// TIA Portal project "Niagara_V1" (V16)

(* hardware
DEVICE "S7-1200 station_1"  S7-1200 Station
   slot 0: "Rack_0"  S7-1200 Rack  Rack  V1.0
   slot 1: "PLC_Start"  CPU 1214C DC/DC/Rly  6ES7 214-1HG40-0XB0  V4.4
   slot 2: "DI 16x24VDC_2"  6ES7 221-1BH32-0XB0  V2.0
   slot 3: "DQ 16xRelay_1"  SM 1222 DQ16 x relay  6ES7 222-1HH32-0XB0  V2.0
   slot 3: "CB 1241 (RS485)"  CB 1241 (RS485)  6ES7 241-1CH30-1XB0  V1.0
   slot 4: "DQ 16xRelay_3"  SM 1222 DQ16 x relay  6ES7 222-1HH32-0XB0  V2.0
   slot 5: "AI 8xRTD_1"  SM 1231 AI8 x RTD  6ES7 231-5PF32-0XB0  V2.0
   slot 6: "AI 4xRTD_1"  SM 1231 AI4 x RTD  6ES7 231-5PD32-0XB0  V2.0
   slot 7: "AQ 4x14BIT_2"  6ES7 232-4HD32-0XB0  V2.1
*)

// ===== PLC "PLC_Start"  CPU 1214C DC/DC/Rly =====

VAR_GLOBAL   // PLC tag table "Default tag table"
   "rAlarm_SetMinPressSteam" AT %MW12 : Int;   // Уставка минимального давления пара
   "rAI_Press1" AT %MW14 : Int;   // Давление датчика
   "bAlarmPress1" AT %M16.0 : Bool;
   "rAlarm_SetMinPressWater" AT %MW18 : Int;   // Уставка аварийного давления воды
   "rAI_Press2" AT %MW20 : Int;
   "test_PID_P_Backup" AT %MD28 : Real;
   "testLoadBackUp" AT %M1.1 : Bool;
   "Test_eee" AT %M1.2 : Bool;
   "System_Byte" AT %MB510 : Byte;
   "FirstScan" AT %M510.0 : Bool;
   "DiagStatusUpdate" AT %M510.1 : Bool;
   "AlwaysTRUE" AT %M510.2 : Bool;
   "AlwaysFALSE" AT %M510.3 : Bool;
END_VAR

VAR_GLOBAL   // PLC tag table "HMI_"
   "bHMI_button_Start" AT %M2.0 : Bool;   // Кнопка старт
   "bHMI_button_Stop" AT %M2.1 : Bool;   // Кнопка стоп
   "bHMI_button_Pause" AT %M2.2 : Bool;   // Кнопка пауза
   "bHMI_Button_ConveyorStart" AT %M2.4 : Bool;   // Кнопка подтверждения старта конвейера
   "bStartAllowed" AT %M100.0 : Bool;   // Готовность к старту
   "bOpenWindStartConveyor" AT %M100.1 : Bool;   // Вызов окна подтверждения оператором старта конвейера
   "iHMI_Num_StatrPaster" AT %MW4 : Int;   // Статус работы пастризаора
   "sHMI_Text_State" AT %MB3 : Char;   // Ткстом статус пастеризатора
   "bTypePID_Zone1" AT %M8.0 : Bool;   // Тип ПИД - 1 - Охлаждение, 0 - Нагрев
   "bTypePID_Zone2" AT %M8.1 : Bool;   // Тип ПИД - 1 - Охлаждение, 0 - Нагрев
   "bTypePID_Zone3" AT %M8.2 : Bool;   // Тип ПИД - 1 - Охлаждение, 0 - Нагрев
   "bTypePID_Zone4" AT %M8.3 : Bool;   // Тип ПИД - 1 - Охлаждение, 0 - Нагрев
   "bTypePID_Zone5" AT %M8.4 : Bool;   // Тип ПИД - 1 - Охлаждение, 0 - Нагрев
   "rHMI_SpeedConveyor" AT %MD60 : Real;   // Расчетная Скорость конвейера
   "rHMI_TimeHoldMin" AT %MD56 : Real;   // Для удобства восприятия времени выдержки
   "bResetCommon" AT %M0.3 : Bool;   // Глобальный сброс аварий
   "bAllAuto" AT %M0.6 : Bool;   // Перевод всего оборудования в авто с ручного
   "bZoomerOff" AT %M0.7 : Bool;   // Выкл пищалка
   "bHMI_button_Start_Sterilization" AT %M2.5 : Bool;   // Кнопка старт Стерилизации
   "bHMI_Steril_Fimish" AT %M8.7 : Bool;   // Стерилизация готова флаг
   "iHMI_Steril_sec" AT %MW22 : Int;   // СЕК таймера стерилизациии
   "iHMI_Steril_min" AT %MW26 : Int;   // МИН таймера стерилизации
   "iHMIWind_FinishStiril" AT %MW32 : Int;   // Всплывающее окно на панели
   "bOpenWindSterilFinish" AT %M34.0 : Bool;   // Вызвать окно окончание стирилизации
   "bHMI_Start_Banya" AT %M8.6 : Bool;   // Кнопка старт режима "Баня"
   "bTypePID_Zone6" AT %M9.1 : Bool;   // Тип ПИД - 1 - Охлаждение, 0 - Нагрев
   "bTypePID_Zone7" AT %M9.2 : Bool;   // Тип ПИД - 1 - Охлаждение, 0 - Нагрев
   "bTypePID_Zone8" AT %M9.3 : Bool;   // Тип ПИД - 1 - Охлаждение, 0 - Нагрев
   "bTypePID_Zone9" AT %M9.4 : Bool;   // Тип ПИД - 1 - Охлаждение, 0 - Нагрев
   "bTypePID_Zone10" AT %M9.5 : Bool;   // Тип ПИД - 1 - Охлаждение, 0 - Нагрев
   "bTypePID_Zone11" AT %M9.6 : Bool;   // Тип ПИД - 1 - Охлаждение, 0 - Нагрев
   "bSafetyMode" AT %M10.3 : Bool;   // Режим защиты от перепастеризации
   "bResSafetyMode" AT %M10.4 : Bool;   // Сброс режима защиты от перепастеризации
   "bCheck_ModeSafety" AT %M10.5 : Bool;   // Галочка - разрешение работы режима защиты от перепастеризации
   "bStateZonesBanya_OK" AT %M10.6 : Bool;   // Статус готовности по зонам в режиме Баня
   "bHasPrior_Stop_Bany" AT %M10.7 : Bool;   // Установлен приоритет по стопу конвейера при отклонении в режиме Баня
   "iNomberZoneAlarmBany" AT %MW40 : Int;   // Номер зоны с отклонениями от уставок
   "rHMI_Fact_SpeedConveyor" AT %MD64 : Real;   // Фактическая Скорость конвейера
END_VAR

VAR_GLOBAL   // PLC tag table "DI"
   "E-Stop №1" AT %I0.0 : Bool;
   "E-Stop №2" AT %I0.1 : Bool;
   "E-Stop №3" AT %I0.2 : Bool;
   "Контроль фаз" AT %I2.7 : Bool;
   "Уровнь_Низ 1" AT %I2.3 : Bool;
   "Уровнь_Верх 1" AT %I2.4 : Bool;
   "Д_Затор" AT %I2.6 : Bool;
   "Частотник (работа) 1" AT %I2.0 : Bool;
   "Частотник (работа) 2" AT %I2.1 : Bool;
   "Частотник (работа) 3" AT %I2.2 : Bool;
   "Пускатель включен 1" AT %I0.3 : Bool;
   "Пускатель включен 2" AT %I0.4 : Bool;
   "Пускатель включен 3" AT %I0.5 : Bool;
   "Пускатель включен 4" AT %I0.6 : Bool;
   "Пускатель включен 5" AT %I0.7 : Bool;
   "Пускатель включен 6" AT %I1.0 : Bool;
   "Пускатель включен 7" AT %I1.1 : Bool;
   "Пускатель включен 8" AT %I1.2 : Bool;
   "Пускатель включен 9" AT %I1.3 : Bool;
   "Пускатель включен 10" AT %I1.4 : Bool;
   "Пускатель вкл Воздуходувка" AT %I1.5 : Bool;
   "Д_Коленвала" AT %I2.5 : Bool;
   "Д_Давл Воздуха" AT %I3.0 : Bool;
END_VAR

VAR_GLOBAL   // PLC tag table "MyTags"
   "rHoldtimeMIN_Out" AT %MD52 : Real;   // Время выдержки в мин
   "Разрешение работы конвейера" AT %M0.0 : Bool;   // Команда разрешения от Глобального блока работы
   "Авария, ошибка в системе" AT %M0.1 : Bool;   // Метка ошибок или аварий
   "iNomberZoneAlarm" AT %MW6 : Int;   // Номер зоны с отклонениями
   "bMain_AlarmSystem" AT %M2.3 : Bool;   // АВария в системе (Общая)
   "bStartWork_Main_TunelPaster" AT %M1.7 : Bool;   // Старт-Работа тунельного пастеризатора (ОБЩИЙ)
   "bHasPrior_Stop" AT %M10.1 : Bool;   // Имеется маркер разрешения "СТОП - конвейер
   "bStateZones_OK" AT %M10.0 : Bool;   // Все зоны готовы к работе
   "bStartFillBac_1" AT %M0.4 : Bool;   // Ком_Наполнение бака 1
   "bStartFillBac_2" AT %M0.5 : Bool;   // Ком_Наполнение бака 2
   "AlarmPress" AT %M0.2 : Bool;   // Общая авария давления
   "bStartWork_Sterilization" AT %M2.6 : Bool;   // Старт-Работа режима стерилизации
   "bState_Stiril_Zone_OK" AT %M1.0 : Bool;   // Все зоны готовы к стерилизации
   "iNumZoneStiril_NotOk" AT %MW24 : Int;   // Номер зоны не готовые стирилизации
   "bStartWork_БАНЯ" AT %M9.0 : Bool;
   "ПЕ_Вер-1" AT %M11.3 : Bool;   // Работа расчета Пе (вер_1)
END_VAR

VAR_GLOBAL   // PLC tag table "Timers_CPU"
   "Time_0.1s" AT %M500.0 : Bool;
   "Time_0.2s" AT %M500.1 : Bool;
   "Time_0.4s" AT %M500.2 : Bool;
   "Time_0.5s" AT %M500.3 : Bool;
   "Time_0.8s" AT %M500.4 : Bool;
   "Time_1s" AT %M500.5 : Bool;
   "Time_1.6s" AT %M500.6 : Bool;
   "Time_2s" AT %M500.7 : Bool;
END_VAR

VAR_GLOBAL   // PLC tag table "DO"
   "Пневмо_остров клапан 1" AT %Q0.0 : Bool;
   "Пневмо_остров клапан 2" AT %Q0.1 : Bool;
   "Пневмо_остров клапан 3" AT %Q0.2 : Bool;
   "Пневмо_остров клапан 4" AT %Q0.3 : Bool;
   "Пневмо_остров клапан 5" AT %Q0.4 : Bool;
   "Пневмо_остров клапан 6" AT %Q0.5 : Bool;
   "Пневмо_остров клапан 7" AT %Q0.6 : Bool;
   "Пневмо_остров клапан 8" AT %Q16.7 : Bool;   // Не используем выход общий с 9 клапаном
   "Пневмо_остров клапан 9" AT %Q1.0 : Bool;
   "Пневмо_остров клапан 10" AT %Q1.1 : Bool;
   "Частотник Пуск 1" AT %Q6.3 : Bool;   // Реле К 9
   "Частотник Пуск 2" AT %Q6.4 : Bool;   // Реле К 10
   "Частотник Пуск 3" AT %Q6.5 : Bool;   // Реле К 11
   "Световая колонна - зеленый" AT %Q7.0 : Bool;
   "Световая колонна - желтый" AT %Q7.1 : Bool;
   "Световая колонна - красный" AT %Q7.2 : Bool;
   "Световая колонна – звуковой сигнал" AT %Q7.3 : Bool;
   "Пускатель №1" AT %Q4.0 : Bool;
   "Пускатель №2" AT %Q4.1 : Bool;
   "Пускатель №3" AT %Q4.2 : Bool;
   "Пускатель №4" AT %Q4.3 : Bool;
   "Пускатель №5" AT %Q4.4 : Bool;
   "Пускатель №6" AT %Q4.5 : Bool;
   "Пускатель №7" AT %Q4.6 : Bool;
   "Пускатель Воздуходувка" AT %Q6.2 : Bool;
   "Пуск транспортера" AT %Q11.0 : Bool;   // Реле К 12
   "Пускатель №8" AT %Q4.7 : Bool;
   "Пускатель №9" AT %Q6.0 : Bool;
   "Пускатель №10" AT %Q6.1 : Bool;
   "Пневмо_остров клапан 11" AT %Q15.0 : Bool;   // Не используем выход общий с 12 клапаном
   "Пневмо_остров клапан 12" AT %Q5.1 : Bool;
   "КЛ_Химия-1" AT %Q5.2 : Bool;
   "КЛ_Пара" AT %Q5.5 : Bool;
   "КЛ_Стирилизации" AT %Q5.6 : Bool;
   "КЛ_Подпидки" AT %Q5.4 : Bool;
   "КЛ_Химия-2" AT %Q5.3 : Bool;
END_VAR

VAR_GLOBAL   // PLC tag table "AI"
   "TT 1" AT %IW140 : Int;   // PT100
   "TT 2" AT %IW142 : Int;   // PT100
   "TT 3" AT %IW144 : Int;   // PT100
   "TT 4" AT %IW146 : Int;   // PT100
   "TT 5" AT %IW148 : Int;   // PT100
   "TT 6" AT %IW150 : Int;   // PT100
   "TT 7" AT %IW152 : Int;   // PT100
   "TT 8" AT %IW154 : Int;   // PT100
   "AI_0.0_Датчик давления 1" AT %IW112 : Int;   // 4-20mA
   "AI_0.1_Датчик давления 2" AT %IW114 : Int;   // 4-20mA
   "AI_0.2_Датчик давления 3" AT %IW116 : Int;   // 4-20mA
   "AI_0.3_" AT %IW118 : Int;   // 4-20mA
   "TT 9" AT %IW156 : Int;
   "TT 10" AT %IW158 : Int;
END_VAR

VAR_GLOBAL   // PLC tag table "AO"
   "Упр частоты 1" AT %QW180 : Int;
   "Упр частоты 2" AT %QW182 : Int;
   "Упр частоты 3" AT %QW184 : Int;
END_VAR

VAR_GLOBAL   // PLC tag table "Alarms"
   "Ai_Alarm_1" AT %M50.0 : Bool;
   "Ai_Alarm_2" AT %M50.1 : Bool;
   "Ai_Alarm_3" AT %M50.2 : Bool;
   "Ai_Alarm_4" AT %M50.3 : Bool;
   "Ai_Alarm_5" AT %M50.4 : Bool;
   "Ai_Alarm_6" AT %M50.5 : Bool;
END_VAR

VAR_GLOBAL   // PLC tag table "__TEST"
   "bT_Alarm" AT %M1.3 : Bool;
   "bTOpenWind" AT %M1.4 : Bool;
   "iTestPause" AT %MW1 : Int;
   "bTZoomOff" AT %M8.5 : Bool;
   "Test_Time" AT %MD36 : DInt;
   "test_reset" AT %M9.7 : Bool;
   "Test_Alarm" AT %M10.2 : Bool;
   "ТестБаня" AT %M11.0 : Bool;
   "ТестБаняОк" AT %M11.1 : Bool;
   "Тест_СтартБаня" AT %M11.2 : Bool;
   "Тест_Старт ПЕ" AT %M11.4 : Bool;
   "Тест-СкоростьКонв" AT %MD42 : Real;
   "T485_MB_ADDR" AT %MW46 : UInt;
   "T485_MODE" AT %MB17 : USInt;
   "T485_DATA_ADDR" AT %MD68 : UDInt;
   "T485_DATA_LEN" AT %MW48 : UInt;
   "T485_GetData" AT %MW11 : Int;
   "T_485_REQ" AT %M16.1 : Bool;
   "MB_ADDR_T1" AT %MW72 : UInt;
   "MB_MODE_T" AT %MB35 : USInt;
   "MB_DATA_ADDR" AT %MD74 : UDInt;
   "MB_LENGH_T" AT %MW78 : UInt;
   "MB_MODE_T2" AT %MB51 : USInt;
   "MB_DATA_ADDR2" AT %MD80 : UDInt;
   "MB_LENGH_T2" AT %MW84 : UInt;
END_VAR

VAR_GLOBAL   // PLC tag table "RS-485"
   "Управляемый клапан №1" AT %MW111 : Int;
   "Управляемый клапан №2" AT %MW114 : Int;
   "Управляемый клапан №3" AT %MW116 : Int;
   "Управляемый клапан №4" AT %MW118 : Int;
   "Управляемый клапан №5" AT %MW120 : Int;
   "Управляемый клапан №6" AT %MW122 : Int;
   "Управляемый клапан №7" AT %MW124 : Int;
   "Управляемый клапан №8" AT %MW126 : Int;
   "Управляемый клапан №9" AT %MW128 : Int;
   "Управляемый клапан №10" AT %MW130 : Int;
   "Управляемый клапан №11" AT %MW132 : Int;
   "Управляемый клапан №12" AT %MW134 : Int;
END_VAR

TYPE "FV_o/c"
   STRUCT
      bOpenCmd : Bool;   // Команда открыть (автомат)
      bManualMode : Bool;   // Ручной режим (TRUE)
      bManualOpen : Bool;   // Команда открыть в ручном режиме
      bFeedbackOpen : Bool;   // Обратная связь "Открыт"
      tMaxTime : Time;   // Время на открытие
      bResetAlarm : Bool;   // Сброс аварии
      bCheckFeedback : Bool;   // Выбирается есть ли обратная связь у клапана
      bOutOpen : Bool;   // Выход на открытие клапана
      iOutState : Int;   // Выход статуса клапана
   END_STRUCT;
END_TYPE

TYPE "ZoneStatus"
   STRUCT
      bInSetpoint : Bool;   // Зона в уставке по температуре
      bOutOfRange : Bool;   // Зона вышла от уставки на > дельта
      bHasPriority : Bool;   // Зона имеет приоритет на остановку конвейера
   END_STRUCT;
END_TYPE

TYPE "Zone_Pararm"
   STRUCT
      rTemp : Real;   // Температура с датчика
      rSet : Real := 20.0;   // Уставка
      rDeltaDown : Real := 1.0;   // ДельтаНижний предел
      rDeltaUP : Real := 1.0;   // ДельтаВерхний Предел
      bPriority : Bool;   // Приоритет
      bOUT_ZoneStatus : "ZoneStatus";   // Состояние зоны_
   END_STRUCT;
END_TYPE

TYPE "FV_regul"
   STRUCT
      bHMI_ManualMode : Bool;   // Переключение режима авто/ручно (0 - А, 1 - Р)
      "bManualOpen/Close" : Bool;   // Ручн режим выход DO для клапана
      rHMI_ManualSet : Real;   // Уставка в ручном режиме (0-100)
      "bAutoOpen/Close" : Bool;   // Авто режим Сигнал DO на выход для клапана
      rAuto_Set : Real;   // Уставка в автоматическом режиме
      iOut_AO : Int;   // Сигнал на аналоговый выход
      "rHMI_Out_FV-%" : Real;   // Состояние в % (0-100)
      "bOut_DO_Open/Close" : Bool;   // Сигнал выход для DO
      bOut_State_ValveOpen : Int;   // Cтатуса - клапан открыт (1)/закрыт(0)
   END_STRUCT;
END_TYPE

TYPE "Коэф ПИД"
   STRUCT
      Set : Real;   // Уставка
      Gain : Int;   // Коэф П
      I : DInt;   // Коэф И
      D : DInt;   // Коэф Д
   END_STRUCT;
END_TYPE

TYPE "PE_Param"
   STRUCT
      rПЕ_Задан : Real;
      rДлина_Конв : Real;
      rZ_Коэф : Real := 1.393;
      rТref : Real := 60.0;
      rТемп_Мин : Real;
      rТемп_Макс : Real;
      "rСкоростьКонв_м/мин" : Real;
      rРучноеЗначТемп : Real;
      diВремяПростоя : DInt := 60000;
      bManualTemp : Bool;
   END_STRUCT;
END_TYPE

TYPE "tipe_Pumps"
   STRUCT
      bAutoMode_Work : Bool;   // автоматический режим
      bManualMode : Bool;   // Ручной режим вкл/выкл
      bManualStart : Bool;   // Старт в ручном режиме
      rManualSpeed : Real;   // Скорость в ручном режиме
      rHMI_Speed : Real;   // Выходная скороость для HMI
      bHMI_PumpRun : Bool;   // Статус работы для HMI
      bresAlarm : Bool;   // Сброс аварий
      iStatusPump : Int;   // Статус насоса
      bIn_DryRunning : Bool;   // Сигнал сухого хода
      bIn_AutomatState : Bool;   // Вход статуса состояния автоматов
      bIn_PuskatelState : Bool;   // Вход статуса состояния пускателя
      bIn_Run_Ok_State : Bool;   // Вход подтверждения старта (частотники)
   END_STRUCT;
END_TYPE

TYPE "Tipe_Conveyor"
   STRUCT
      bManualMode : Bool;   // Ручной режим вкл/выкл
      bManualStart : Bool;   // Старт в ручном режиме
      rManualSpeed : Real;   // Скорость в ручном режиме
      bresAlarm : Bool;   // Сброс аварий
      rAutoSpeed : Real;   // Автомат_Заданная скорость конвеера
      rHMI_Speed : Real;   // Выходная скороость для HMI
      bHMI_Conv_Run : Bool;   // Статус работы для HMI
      iStatusConve : Int;   // Статус конвейера
      bIn_AutomatState : Bool;   // Вход статуса состояния автоматов
      bInPuskatelState : Bool;   // Вход статуса состояния пускателя
      bInRun_Ok_State : Bool;   // Вход подтверждения старта (частотники)
   END_STRUCT;
END_TYPE

TYPE "Tipe_DI"
   STRUCT
      f_DI_out : Bool;
      "bFiltr_on/off" : Bool := true;   // Вкл/выкл фильтрацию входа
      diTime_filtr : Time := T#100ms;   // Уставка времени фильтрации
      bSimulation : Bool;   // Включение режима симуляции
      "bSim_On/Off" : Bool;   // Управление симуляцией
   END_STRUCT;
END_TYPE

TYPE "Tipe_Filling_Bac"
   STRUCT
      bManualMode : Bool;
      bManualOpen : Bool;
      diTimeCloseValve : DInt;   // Таймер задержки закрытия клапана по верхнему уровню
   END_STRUCT;
END_TYPE

TYPE "Tipe_AI"
   STRUCT
      bSimulate : Bool;   // Вкл симуляции датчика
      rSimulateValue : Real;   // Значение симуляции датчика
      rSensor_HL : Real;   // Верхний предел датчика
      rSensor_LL : Real;   // Нижний предел датчика
      bFiltr : Bool;   // Управление фильтром значений
      rAI_Value : Real;   // Значение аналогового датчика
   END_STRUCT;
END_TYPE

TYPE "tipePress"
   STRUCT
      rInPress : Real;   // Значение с датчика
      rSetpoint : Real := 2.0;   // Уставка минимального давления
      bAlarm_Press : Bool;   // Выход АВАРИЯ
   END_STRUCT;
END_TYPE

TYPE "tipePumpHim"
   STRUCT
      Чек_вРежимеПастер : Bool;   // Указание в панели на разрешения работы насоса в режиме пастеризации
      Чек_вРежимеМойка : Bool;   // Указание в панели на разрешения работы насоса в режиме Мойка
      ВремяРаботы : DInt := 5;   // Время продолжительности импульса работы насоса
      ВремяПаузы : DInt := 10;   // Время паузы между импульсами
   END_STRUCT;
END_TYPE

TYPE "StopMgr"
   STRUCT
      Timer_Stop : IEC_TIMER;   // Таймер длительности простоя
      Duration : Time;   // Длительность простоя
      PU_Stop_Add : Real;   // Доп. ПЕ, набранные на простое
      Reject_Required : Bool;   // Флаг необходимости отбраковки
   END_STRUCT;
END_TYPE

// folder: PE_V2

TYPE "Zone_Config"
   STRUCT
      Length : Real;   // Длина зоны (м)
      TempWater_Set : Real;   // Уставка температуры воды (°C)
      TempWater_Act : Real;   // Фактическая температура воды (°C)
      TimeInZone : Real;   // Расчётное время в зоне (мин)
      TempProd_In : Real;   // Т-ра продукта на входе в зону (°C)
      TempProd_Out : Real;   // Т-ра продукта на выходе из зоны (°C)
      TempProd_Avg : Real;   // Средняя Т-ра в зоне (°C)
      PU_Zone : Real;   // ПЕ, накопленные в этой зоне
      ZoneType : Bool;   // 1=Нагрев, 2=Выдержка, 3=Охлаждение
      Status_OK : Bool;   // Флаг: расчёт корректен
   END_STRUCT;
END_TYPE

TYPE "ProductPosition"
   STRUCT
      TempProduct : Real;   // Расчётная температура продукта (°C)
      PU_Accumulated : Real;   // Накопленные ПЕ для этой позиции
      InTunnel : Bool;   // Флаг: позиция занята продуктом
      ZoneIndex : Int;   // Номер текущей зоны (1-9)
   END_STRUCT;
END_TYPE

TYPE "Recipe"
   STRUCT
      ID : Int;   // ID рецепта
      "Name" : String;   // Название рецепта
      K_Coeff : Real;   // Коэффициент теплопередачи (1/мин)
      PU_Target_Min : Real;   // Минимально допустимые ПЕ
      PU_Target_Max : Real;   // Максимально допустимые ПЕ
      TempProd_Inlet : Real;   // Температура продукта на входе (°C)
      Speed_Set : Real;   // Уставка скорости ленты (м/мин)
      ZoneConfig : Array[1..9] of "Zone_Config";   // Массив зон
   END_STRUCT;
END_TYPE

TYPE "Status_V2"
   STRUCT
      PU_Total : Real;   // Итоговые ПЕ (последняя вышедшая бутылка)
      PU_Current_Avg : Real;   // Средние ПЕ продукта сейчас в туннеле
      TempProd_Max : Real;   // Макс. температура продукта в туннеле
      Speed_Act : Real;   // Фактическая скорость (м/мин)
      PosCount : Int;   // Количество активных позиций в туннеле
      Line_Run : Bool;   // Статус линии (1=работает)
   END_STRUCT;
END_TYPE

TYPE "Alarm"
   STRUCT
      Temp_Deviation : Bool;   // Отклонение температуры воды
      PU_Under : Bool;   // Недопастеризация
      PU_Over : Bool;   // Перепастеризация
      Sensor_Fault : Bool;   // Неисправность датчика
      Stop_Request : Bool;   // Запрос остановки линии
      Jam_Detected : Bool;   // Сигнал затора
   END_STRUCT;
END_TYPE

// folder: PE_V3

TYPE "ZoneDate"
   STRUCT
      TempWater_Act : Real;   // Фактическая температура воды (°C)
      TimeInZone : Real;   // Расчётное время в зоне (мин)
      TempProd_In : Real;   // Т-ра продукта на входе в зону (°C)
      TempProd_Out : Real;   // Т-ра продукта на выходе из зоны (°C)
      TempProd_Avg : Real;   // Средняя Т-ра в зоне (°C)
      PU_Zone : Real;   // ПЕ, накопленные в этой зоне
   END_STRUCT;
END_TYPE

TYPE "Status_V3"
   STRUCT
      PU_Total : Real;   // Итоговые ПЕ (последняя вышедшая бутылка)
      TempProd_Exit : Real;
      Speed_Act : Real;   // Фактическая скорость (м/мин)
      Line_Run : Bool;   // Статус линии (1=работает)
      ZoneData : Array[1..9] of "ZoneDate";   // Данные по зонам
      Calculation_Ready : Bool;   // Флаг: расчёт выполнен
   END_STRUCT;
END_TYPE

TYPE "Zone_Config_V3"
   STRUCT
      Length : Real;   // Длина зоны (м)
      TempWater_Set : Real;   // Уставка температуры воды (°C)
   END_STRUCT;
END_TYPE

// folder: (top level)

DATA_BLOCK "Test_Beep_DB"   // DB129
{ S7_Optimized_Access := 'TRUE' }
VERSION : 0.1
// stored: InstanceOfName Test_Beep
"Test_Beep"
BEGIN
END_DATA_BLOCK

DATA_BLOCK "Расчет ПЕ по сек_DB"   // DB178
{ S7_Optimized_Access := 'TRUE' }
VERSION : 0.1
// stored: InstanceOfName Расчет ПЕ по сек
"Расчет ПЕ по сек"
BEGIN
END_DATA_BLOCK

DATA_BLOCK "Расчет ПЕ по Зонам(aver)_DB"   // DB180
{ S7_Optimized_Access := 'TRUE' }
VERSION : 0.1
// stored: InstanceOfName Расчет ПЕ по Зонам(aver)
"Расчет ПЕ по Зонам(aver)"
BEGIN
END_DATA_BLOCK

DATA_BLOCK "Расчет ПЕ по Зонам(aver) -Расчетное_DB"   // DB181
{ S7_Optimized_Access := 'TRUE' }
VERSION : 0.1
// stored: InstanceOfName Расчет ПЕ по Зонам(aver)
"Расчет ПЕ по Зонам(aver)"
BEGIN
END_DATA_BLOCK

DATA_BLOCK "Test_RS485"   // DB194
{ S7_Optimized_Access := 'FALSE' }
VERSION : 0.1
   VAR
      in : Array[0..315] of Int;
      Out_Set : UInt;
   END_VAR
BEGIN
END_DATA_BLOCK

DATA_BLOCK "Regul_FV_RS485"   // DB195
{ S7_Optimized_Access := 'FALSE' }
VERSION : 0.1
   VAR
      Set_FV : Array[1..12] of Int;
   END_VAR
BEGIN
END_DATA_BLOCK

// folder: AI_Signal/AI_DB/PT100

DATA_BLOCK "AI_1_(PT100)_DB"   // DB88
{ S7_Optimized_Access := 'FALSE' }
VERSION : 0.1
// stored: InstanceOfName AI_(PT100)
"AI_(PT100)"
BEGIN
END_DATA_BLOCK

DATA_BLOCK "AI_2_(PT100)_DB"   // DB89
{ S7_Optimized_Access := 'FALSE' }
VERSION : 0.1
// stored: InstanceOfName AI_(PT100)
"AI_(PT100)"
BEGIN
END_DATA_BLOCK

DATA_BLOCK "AI_3_(PT100)_DB"   // DB91
{ S7_Optimized_Access := 'FALSE' }
VERSION : 0.1
// stored: InstanceOfName AI_(PT100)
"AI_(PT100)"
BEGIN
END_DATA_BLOCK

DATA_BLOCK "AI_4_(PT100)_DB"   // DB92
{ S7_Optimized_Access := 'FALSE' }
VERSION : 0.1
// stored: InstanceOfName AI_(PT100)
"AI_(PT100)"
BEGIN
END_DATA_BLOCK

DATA_BLOCK "AI_5_(PT100)_DB"   // DB93
{ S7_Optimized_Access := 'FALSE' }
VERSION : 0.1
// stored: InstanceOfName AI_(PT100)
"AI_(PT100)"
BEGIN
END_DATA_BLOCK

DATA_BLOCK "AI_6_(PT100)_DB"   // DB112
{ S7_Optimized_Access := 'FALSE' }
VERSION : 0.1
// stored: InstanceOfName AI_(PT100)
"AI_(PT100)"
BEGIN
END_DATA_BLOCK

DATA_BLOCK "AI_7_(PT100)_DB"   // DB113
{ S7_Optimized_Access := 'FALSE' }
VERSION : 0.1
// stored: InstanceOfName AI_(PT100)
"AI_(PT100)"
BEGIN
END_DATA_BLOCK

// folder: DB-FB

DATA_BLOCK "FB_check_For_Start_Paster_DB"   // DB1
{ S7_Optimized_Access := 'FALSE' }
VERSION : 0.1
// stored: InstanceOfName FB_check_For_Start
"FB_check_For_Start"
BEGIN
END_DATA_BLOCK

DATA_BLOCK "FB_Emergency_DB"   // DB3
{ S7_Optimized_Access := 'FALSE' }
VERSION : 0.1
// stored: InstanceOfName FB_Аварии
"FB_Аварии"
BEGIN
END_DATA_BLOCK

DATA_BLOCK "FB_CheckZoneStatus_DB"   // DB11
{ S7_Optimized_Access := 'FALSE' }
VERSION : 0.1
// stored: InstanceOfName FB_CheckZoneStatus
"FB_CheckZoneStatus"
BEGIN
END_DATA_BLOCK

DATA_BLOCK "FB_Управление конвейером_DB"   // DB18
{ S7_Optimized_Access := 'FALSE' }
VERSION : 0.1
// stored: InstanceOfName FB_Управление конвейером
"FB_Управление конвейером"
BEGIN
END_DATA_BLOCK

DATA_BLOCK "FB_GlobalStateManager_DB"   // DB31
{ S7_Optimized_Access := 'FALSE' }
VERSION : 0.1
// stored: InstanceOfName FB_GlobalStateManager
"FB_GlobalStateManager"
BEGIN
END_DATA_BLOCK

DATA_BLOCK "FB_PE_Control_DB"   // DB38
{ S7_Optimized_Access := 'TRUE' }
VERSION : 0.1
// stored: InstanceOfName FB_ПЕ_Control
"FB_ПЕ_Control"
BEGIN
END_DATA_BLOCK

DATA_BLOCK "Главный блок конвейера_DB"   // DB39
{ S7_Optimized_Access := 'TRUE' }
VERSION : 0.1
// stored: InstanceOfName FB_Главный блок конвейера
"FB_Главный блок конвейера"
BEGIN
END_DATA_BLOCK

DATA_BLOCK "R_trig_All_Auto"   // DB40
{ S7_Optimized_Access := 'TRUE' }
VERSION : 0.1
// stored: InstanceOfName R_trig
"R_trig"
BEGIN
END_DATA_BLOCK

DATA_BLOCK "FB_Sterilization_CheckZoneStatus_DB"   // DB41
{ S7_Optimized_Access := 'FALSE' }
VERSION : 0.1
// stored: InstanceOfName FB_Stiril_CheckZoneStatus
"FB_Stiril_CheckZoneStatus"
BEGIN
END_DATA_BLOCK

DATA_BLOCK "FB_Steril_Timer_DB"   // DB42
{ S7_Optimized_Access := 'TRUE' }
VERSION : 0.1
// stored: InstanceOfName FB_Steril_Timer
"FB_Steril_Timer"
BEGIN
END_DATA_BLOCK

DATA_BLOCK "Вентилятор_DB"   // DB46
{ S7_Optimized_Access := 'FALSE' }
VERSION : 0.1
// stored: InstanceOfName Pump
"Pump"
BEGIN
END_DATA_BLOCK

DATA_BLOCK "FB_Mode_Paster_DB"   // DB81
{ S7_Optimized_Access := 'TRUE' }
VERSION : 0.1
// stored: InstanceOfName FB_Mode_Paster
"FB_Mode_Paster"
BEGIN
END_DATA_BLOCK

DATA_BLOCK "FB_Filling_Bac1_DB"   // DB84
{ S7_Optimized_Access := 'TRUE' }
VERSION : 0.1
// stored: InstanceOfName FB_Filling_Bac
"FB_Filling_Bac"
BEGIN
END_DATA_BLOCK

DATA_BLOCK "FB_Filling_Bac2_DB"   // DB86
{ S7_Optimized_Access := 'TRUE' }
VERSION : 0.1
// stored: InstanceOfName FB_Filling_Bac
"FB_Filling_Bac"
BEGIN
END_DATA_BLOCK

DATA_BLOCK "FB_Press_Controll_Water_DB"   // DB96
{ S7_Optimized_Access := 'TRUE' }
VERSION : 0.1
// stored: InstanceOfName FB_Press_Controll
"FB_Press_Controll"
BEGIN
END_DATA_BLOCK

DATA_BLOCK "FB_Press_Controll_Steam_DB"   // DB97
{ S7_Optimized_Access := 'TRUE' }
VERSION : 0.1
// stored: InstanceOfName FB_Press_Controll
"FB_Press_Controll"
BEGIN
END_DATA_BLOCK

DATA_BLOCK "FB_Press_Controll_Glikol_DB"   // DB98
{ S7_Optimized_Access := 'TRUE' }
VERSION : 0.1
// stored: InstanceOfName FB_Press_Controll
"FB_Press_Controll"
BEGIN
END_DATA_BLOCK

DATA_BLOCK "R_trig_DB"   // DB99
{ S7_Optimized_Access := 'TRUE' }
VERSION : 0.1
// stored: InstanceOfName R_trig
"R_trig"
BEGIN
END_DATA_BLOCK

DATA_BLOCK "R_trig_DB_Alarm_Zoomer"   // DB101
{ S7_Optimized_Access := 'TRUE' }
VERSION : 0.1
// stored: InstanceOfName R_trig
"R_trig"
BEGIN
END_DATA_BLOCK

DATA_BLOCK "FB_SVETOFOR_DB"   // DB102
{ S7_Optimized_Access := 'TRUE' }
VERSION : 0.1
// stored: InstanceOfName FB_SVETOFOR
"FB_SVETOFOR"
BEGIN
END_DATA_BLOCK

DATA_BLOCK "FB_check_For_Start_Sterilization_DB"   // DB103
{ S7_Optimized_Access := 'FALSE' }
VERSION : 0.1
// stored: InstanceOfName FB_check_For_Start
"FB_check_For_Start"
BEGIN
END_DATA_BLOCK

DATA_BLOCK "FB_STIRIL_Mode_DB"   // DB115
{ S7_Optimized_Access := 'TRUE' }
VERSION : 0.1
// stored: InstanceOfName FB_Mode_STIRIL
"FB_Mode_STIRIL"
BEGIN
END_DATA_BLOCK

DATA_BLOCK "FB_Mode_Bany_DB"   // DB122
{ S7_Optimized_Access := 'TRUE' }
VERSION : 0.1
// stored: InstanceOfName FB_Mode_Bany
"FB_Mode_Bany"
BEGIN
END_DATA_BLOCK

DATA_BLOCK "R_trig_OpenWindOper"   // DB124
{ S7_Optimized_Access := 'TRUE' }
VERSION : 0.1
// stored: InstanceOfName R_trig
"R_trig"
BEGIN
END_DATA_BLOCK

DATA_BLOCK "R_trig_Puasa"   // DB125
{ S7_Optimized_Access := 'TRUE' }
VERSION : 0.1
// stored: InstanceOfName R_trig
"R_trig"
BEGIN
END_DATA_BLOCK

DATA_BLOCK "FB_check_For_Start_Banya_DB"   // DB152
{ S7_Optimized_Access := 'FALSE' }
VERSION : 0.1
// stored: InstanceOfName FB_check_For_Start
"FB_check_For_Start"
BEGIN
END_DATA_BLOCK

DATA_BLOCK "FB_Защита от Перепастеризации_DB"   // DB157
{ S7_Optimized_Access := 'TRUE' }
VERSION : 0.1
// stored: InstanceOfName FB_Защита от Перепастеризации
"FB_Защита от Перепастеризации"
BEGIN
END_DATA_BLOCK

DATA_BLOCK "FB_CheckZoneStatus_Bany_DB"   // DB164
{ S7_Optimized_Access := 'FALSE' }
VERSION : 0.1
// stored: InstanceOfName FB_CheckZoneStatus
"FB_CheckZoneStatus"
BEGIN
END_DATA_BLOCK

DATA_BLOCK "FB_Расчет скорости по импульсам_DB"   // DB165
{ S7_Optimized_Access := 'TRUE' }
VERSION : 0.1
// stored: InstanceOfName FB_Расчет скорости по импульсам
"FB_Расчет скорости по импульсам"
BEGIN
END_DATA_BLOCK

// folder: DB_Convert_Rs485

DATA_BLOCK "FB_Convert_For_RS485_7_DB"   // DB197
{ S7_Optimized_Access := 'TRUE' }
VERSION : 0.1
// stored: InstanceOfName FB_Convert_For_RS485
"FB_Convert_For_RS485"
BEGIN
END_DATA_BLOCK

DATA_BLOCK "FB_Convert_For_RS485_2_DB"   // DB199
{ S7_Optimized_Access := 'TRUE' }
VERSION : 0.1
// stored: InstanceOfName FB_Convert_For_RS485
"FB_Convert_For_RS485"
BEGIN
END_DATA_BLOCK

DATA_BLOCK "FB_Convert_For_RS485_1_DB"   // DB200
{ S7_Optimized_Access := 'TRUE' }
VERSION : 0.1
// stored: InstanceOfName FB_Convert_For_RS485
"FB_Convert_For_RS485"
BEGIN
END_DATA_BLOCK

DATA_BLOCK "FB_Convert_For_RS485_3_DB"   // DB201
{ S7_Optimized_Access := 'TRUE' }
VERSION : 0.1
// stored: InstanceOfName FB_Convert_For_RS485
"FB_Convert_For_RS485"
BEGIN
END_DATA_BLOCK

DATA_BLOCK "FB_Convert_For_RS485_4_DB"   // DB202
{ S7_Optimized_Access := 'TRUE' }
VERSION : 0.1
// stored: InstanceOfName FB_Convert_For_RS485
"FB_Convert_For_RS485"
BEGIN
END_DATA_BLOCK

DATA_BLOCK "FB_Convert_For_RS485_5_DB"   // DB203
{ S7_Optimized_Access := 'TRUE' }
VERSION : 0.1
// stored: InstanceOfName FB_Convert_For_RS485
"FB_Convert_For_RS485"
BEGIN
END_DATA_BLOCK

DATA_BLOCK "FB_Convert_For_RS485_6_DB"   // DB204
{ S7_Optimized_Access := 'TRUE' }
VERSION : 0.1
// stored: InstanceOfName FB_Convert_For_RS485
"FB_Convert_For_RS485"
BEGIN
END_DATA_BLOCK

DATA_BLOCK "FB_Convert_For_RS485_8_DB"   // DB205
{ S7_Optimized_Access := 'TRUE' }
VERSION : 0.1
// stored: InstanceOfName FB_Convert_For_RS485
"FB_Convert_For_RS485"
BEGIN
END_DATA_BLOCK

DATA_BLOCK "FB_Convert_For_RS485_9_DB"   // DB206
{ S7_Optimized_Access := 'TRUE' }
VERSION : 0.1
// stored: InstanceOfName FB_Convert_For_RS485
"FB_Convert_For_RS485"
BEGIN
END_DATA_BLOCK

DATA_BLOCK "FB_Convert_For_RS485_10_DB"   // DB207
{ S7_Optimized_Access := 'TRUE' }
VERSION : 0.1
// stored: InstanceOfName FB_Convert_For_RS485
"FB_Convert_For_RS485"
BEGIN
END_DATA_BLOCK

DATA_BLOCK "FB_Convert_For_RS485_11_DB"   // DB208
{ S7_Optimized_Access := 'TRUE' }
VERSION : 0.1
// stored: InstanceOfName FB_Convert_For_RS485
"FB_Convert_For_RS485"
BEGIN
END_DATA_BLOCK

DATA_BLOCK "FB_Convert_For_RS485_12_DB"   // DB209
{ S7_Optimized_Access := 'TRUE' }
VERSION : 0.1
// stored: InstanceOfName FB_Convert_For_RS485
"FB_Convert_For_RS485"
BEGIN
END_DATA_BLOCK

// folder: DI_signal/DB_DI

DATA_BLOCK "DI_EStop1"   // DB48
{ S7_Optimized_Access := 'FALSE' }
VERSION : 0.1
// stored: InstanceOfName FB_DI
"FB_DI"
BEGIN
END_DATA_BLOCK

DATA_BLOCK "DI_EStop2"   // DB49
{ S7_Optimized_Access := 'FALSE' }
VERSION : 0.1
// stored: InstanceOfName FB_DI
"FB_DI"
BEGIN
END_DATA_BLOCK

DATA_BLOCK "DI_EStop3"   // DB50
{ S7_Optimized_Access := 'FALSE' }
VERSION : 0.1
// stored: InstanceOfName FB_DI
"FB_DI"
BEGIN
END_DATA_BLOCK

DATA_BLOCK "DI_ReleVolt"   // DB51
{ S7_Optimized_Access := 'FALSE' }
VERSION : 0.1
// stored: InstanceOfName FB_DI
"FB_DI"
BEGIN
END_DATA_BLOCK

DATA_BLOCK "DI_1_Уровень_Низ"   // DB52
{ S7_Optimized_Access := 'FALSE' }
VERSION : 0.1
// stored: InstanceOfName FB_DI
"FB_DI"
BEGIN
END_DATA_BLOCK

DATA_BLOCK "DI_1_Уровень_Верх"   // DB53
{ S7_Optimized_Access := 'FALSE' }
VERSION : 0.1
// stored: InstanceOfName FB_DI
"FB_DI"
BEGIN
END_DATA_BLOCK

DATA_BLOCK "DI_2_Уровень_Низ"   // DB54
{ S7_Optimized_Access := 'FALSE' }
VERSION : 0.1
// stored: InstanceOfName FB_DI
"FB_DI"
BEGIN
END_DATA_BLOCK

DATA_BLOCK "DI_2_Уровень_Верх"   // DB55
{ S7_Optimized_Access := 'FALSE' }
VERSION : 0.1
// stored: InstanceOfName FB_DI
"FB_DI"
BEGIN
END_DATA_BLOCK

DATA_BLOCK "DI_Индуктивный датчик конв - 1"   // DB56
{ S7_Optimized_Access := 'FALSE' }
VERSION : 0.1
// stored: InstanceOfName FB_DI
"FB_DI"
BEGIN
END_DATA_BLOCK

DATA_BLOCK "DI_Индуктивный датчик конв - 2"   // DB57
{ S7_Optimized_Access := 'FALSE' }
VERSION : 0.1
// stored: InstanceOfName FB_DI
"FB_DI"
BEGIN
END_DATA_BLOCK

DATA_BLOCK "DI_Частотник_1_Готов"   // DB58
{ S7_Optimized_Access := 'FALSE' }
VERSION : 0.1
// stored: InstanceOfName FB_DI
"FB_DI"
BEGIN
END_DATA_BLOCK

DATA_BLOCK "DI_Частотник_2_Готов"   // DB59
{ S7_Optimized_Access := 'FALSE' }
VERSION : 0.1
// stored: InstanceOfName FB_DI
"FB_DI"
BEGIN
END_DATA_BLOCK

DATA_BLOCK "DI_Частотник_3_Готов"   // DB60
{ S7_Optimized_Access := 'FALSE' }
VERSION : 0.1
// stored: InstanceOfName FB_DI
"FB_DI"
BEGIN
END_DATA_BLOCK

DATA_BLOCK "DI_Частотник_4_Готов"   // DB61
{ S7_Optimized_Access := 'FALSE' }
VERSION : 0.1
// stored: InstanceOfName FB_DI
"FB_DI"
BEGIN
END_DATA_BLOCK

DATA_BLOCK "DI_Мотор-Автомат-1(вкл)"   // DB62
{ S7_Optimized_Access := 'FALSE' }
VERSION : 0.1
// stored: InstanceOfName FB_DI
"FB_DI"
BEGIN
END_DATA_BLOCK

DATA_BLOCK "DI_Мотор-Автомат-2(вкл)"   // DB63
{ S7_Optimized_Access := 'FALSE' }
VERSION : 0.1
// stored: InstanceOfName FB_DI
"FB_DI"
BEGIN
END_DATA_BLOCK

DATA_BLOCK "DI_Мотор-Автомат-3(вкл)"   // DB64
{ S7_Optimized_Access := 'FALSE' }
VERSION : 0.1
// stored: InstanceOfName FB_DI
"FB_DI"
BEGIN
END_DATA_BLOCK

DATA_BLOCK "DI_Мотор-Автомат-4(вкл)"   // DB65
{ S7_Optimized_Access := 'FALSE' }
VERSION : 0.1
// stored: InstanceOfName FB_DI
"FB_DI"
BEGIN
END_DATA_BLOCK

DATA_BLOCK "DI_Мотор-Автомат-5(вкл)"   // DB66
{ S7_Optimized_Access := 'FALSE' }
VERSION : 0.1
// stored: InstanceOfName FB_DI
"FB_DI"
BEGIN
END_DATA_BLOCK

DATA_BLOCK "DI_Мотор-Автомат-6(вкл)"   // DB67
{ S7_Optimized_Access := 'FALSE' }
VERSION : 0.1
// stored: InstanceOfName FB_DI
"FB_DI"
BEGIN
END_DATA_BLOCK

DATA_BLOCK "DI_Мотор-Автомат-7(вкл)"   // DB68
{ S7_Optimized_Access := 'FALSE' }
VERSION : 0.1
// stored: InstanceOfName FB_DI
"FB_DI"
BEGIN
END_DATA_BLOCK

DATA_BLOCK "DI_Мотор-Автомат-8(вкл)"   // DB69
{ S7_Optimized_Access := 'FALSE' }
VERSION : 0.1
// stored: InstanceOfName FB_DI
"FB_DI"
BEGIN
END_DATA_BLOCK

DATA_BLOCK "DI_Мотор-Автомат-9(вкл)"   // DB70
{ S7_Optimized_Access := 'FALSE' }
VERSION : 0.1
// stored: InstanceOfName FB_DI
"FB_DI"
BEGIN
END_DATA_BLOCK

DATA_BLOCK "DI_Мотор-Автомат-10(вкл)"   // DB71
{ S7_Optimized_Access := 'FALSE' }
VERSION : 0.1
// stored: InstanceOfName FB_DI
"FB_DI"
BEGIN
END_DATA_BLOCK

DATA_BLOCK "DI_Пускатель - 1(вкл)"   // DB72
{ S7_Optimized_Access := 'FALSE' }
VERSION : 0.1
// stored: InstanceOfName FB_DI
"FB_DI"
BEGIN
END_DATA_BLOCK

DATA_BLOCK "DI_Пускатель - 2(вкл)"   // DB73
{ S7_Optimized_Access := 'FALSE' }
VERSION : 0.1
// stored: InstanceOfName FB_DI
"FB_DI"
BEGIN
END_DATA_BLOCK

DATA_BLOCK "DI_Пускатель - 3(вкл)"   // DB74
{ S7_Optimized_Access := 'FALSE' }
VERSION : 0.1
// stored: InstanceOfName FB_DI
"FB_DI"
BEGIN
END_DATA_BLOCK

DATA_BLOCK "DI_Пускатель - 4(вкл)"   // DB75
{ S7_Optimized_Access := 'FALSE' }
VERSION : 0.1
// stored: InstanceOfName FB_DI
"FB_DI"
BEGIN
END_DATA_BLOCK

DATA_BLOCK "DI_Пускатель - 5(вкл)"   // DB76
{ S7_Optimized_Access := 'FALSE' }
VERSION : 0.1
// stored: InstanceOfName FB_DI
"FB_DI"
BEGIN
END_DATA_BLOCK

DATA_BLOCK "DI_Пускатель - 6(вкл)"   // DB77
{ S7_Optimized_Access := 'FALSE' }
VERSION : 0.1
// stored: InstanceOfName FB_DI
"FB_DI"
BEGIN
END_DATA_BLOCK

DATA_BLOCK "DI_Мотор-Автомат-11(вкл)"   // DB116
{ S7_Optimized_Access := 'FALSE' }
VERSION : 0.1
// stored: InstanceOfName FB_DI
"FB_DI"
BEGIN
END_DATA_BLOCK

DATA_BLOCK "DI_Пускатель - 7(вкл)"   // DB117
{ S7_Optimized_Access := 'FALSE' }
VERSION : 0.1
// stored: InstanceOfName FB_DI
"FB_DI"
BEGIN
END_DATA_BLOCK

DATA_BLOCK "DI_Пускатель - 8(вкл)"   // DB118
{ S7_Optimized_Access := 'FALSE' }
VERSION : 0.1
// stored: InstanceOfName FB_DI
"FB_DI"
BEGIN
END_DATA_BLOCK

DATA_BLOCK "DI_Пускатель - 9(вкл)"   // DB167
{ S7_Optimized_Access := 'FALSE' }
VERSION : 0.1
// stored: InstanceOfName FB_DI
"FB_DI"
BEGIN
END_DATA_BLOCK

DATA_BLOCK "DI_Пускатель - 10(вкл)"   // DB168
{ S7_Optimized_Access := 'FALSE' }
VERSION : 0.1
// stored: InstanceOfName FB_DI
"FB_DI"
BEGIN
END_DATA_BLOCK

DATA_BLOCK "DI_Пускатель - Воздуходувка(вкл)"   // DB169
{ S7_Optimized_Access := 'FALSE' }
VERSION : 0.1
// stored: InstanceOfName FB_DI
"FB_DI"
BEGIN
END_DATA_BLOCK

DATA_BLOCK "DI_V_Conveer"   // DB170
{ S7_Optimized_Access := 'FALSE' }
VERSION : 0.1
// stored: InstanceOfName FB_DI
"FB_DI"
BEGIN
END_DATA_BLOCK

// folder: System blocks/Program resources

DATA_BLOCK "IEC_Timer_0_DB"   // DB44
{ S7_Optimized_Access := 'TRUE' }
AUTHOR : Simatic
FAMILY : IEC
NAME : IEC_TMR
VERSION : 1.0
// stored: InstanceOfName IEC_TIMER
"IEC_TIMER"
BEGIN
END_DATA_BLOCK

DATA_BLOCK "IEC_Timer_0_DB_1"   // DB45
{ S7_Optimized_Access := 'TRUE' }
AUTHOR : Simatic
FAMILY : IEC
NAME : IEC_TMR
VERSION : 1.0
// stored: InstanceOfName IEC_TIMER
"IEC_TIMER"
BEGIN
END_DATA_BLOCK

DATA_BLOCK "IEC_Timer_0_DB_3"   // DB47
{ S7_Optimized_Access := 'TRUE' }
AUTHOR : Simatic
FAMILY : IEC
NAME : IEC_TMR
VERSION : 1.0
// stored: InstanceOfName IEC_TIMER
"IEC_TIMER"
BEGIN
END_DATA_BLOCK

DATA_BLOCK "IEC_Timer_0_DB_2"   // DB100
{ S7_Optimized_Access := 'TRUE' }
AUTHOR : Simatic
FAMILY : IEC
NAME : IEC_TMR
VERSION : 1.0
// stored: InstanceOfName IEC_TIMER
"IEC_TIMER"
BEGIN
END_DATA_BLOCK

DATA_BLOCK "IEC_Timer_0_DB_5"   // DB121
{ S7_Optimized_Access := 'TRUE' }
AUTHOR : Simatic
FAMILY : IEC
NAME : IEC_TMR
VERSION : 1.0
// stored: InstanceOfName IEC_TIMER
"IEC_TIMER"
BEGIN
END_DATA_BLOCK

DATA_BLOCK "IEC_Timer_0_DB_11"   // DB123
{ S7_Optimized_Access := 'TRUE' }
AUTHOR : Simatic
FAMILY : IEC
NAME : IEC_TMR
VERSION : 1.0
// stored: InstanceOfName IEC_TIMER
"IEC_TIMER"
BEGIN
END_DATA_BLOCK

DATA_BLOCK "RS485_Counter_0_DB"   // DB196
{ S7_Optimized_Access := 'TRUE' }
AUTHOR : Simatic
FAMILY : IEC
NAME : CNTR
VERSION : 1.0
// stored: InstanceOfName IEC_COUNTER
"IEC_COUNTER"
BEGIN
END_DATA_BLOCK

// folder: Use VARs to HMI

DATA_BLOCK "DB2_HMI_SET"   // DB2
{ S7_Optimized_Access := 'FALSE' }
VERSION : 0.1
   VAR
      dwSetMinWaitGoPause : DInt := 1;   // Время ожидания при выходе за пределы уставок
      dwSetMinWaitComeToGo : DInt := 1;   // Время ожидания при возврате к уставкам
      dwSetTimeWaitToStart : DInt := 60;   // Время ожидания выхода на режим пастеризатора
      dwSetTimeWaitToSPause : DInt := 60;   // Время ожидания Нахождения в паузе
      iTime_Steriliz : Int := 10;   // Время стерилизации
      diTimeHim_1_Paster : DInt := 10;   // Время работы хим насоса-1 в режиме Пастер
      diTimeHim_1_CIP : DInt := 10;   // Время работы хим насоса-1 в режиме Мойка
      diTimePauseHim_1_Paster_1 : DInt := 10;   // Пауза между работой насосов
      diTimePauseHim_1_CIP_1 : DInt := 10;
      diTimeHim_2_Paster : DInt := 10;   // Время работы хим насоса-2 в режиме Пастер
      diTimeHim_2_CIP : DInt := 10;   // Время работы хим насоса-2 в режиме Мойка
      diTimePauseHim_2_Paster : DInt := 10;   // Пауза между работой насосов
      diTimePauseHim_2_CIP : DInt := 10;
      diTimeSafetyModeWait : DInt := 30;   // Время перехода в режим защиты от перепастеризации
   END_VAR
BEGIN
END_DATA_BLOCK

DATA_BLOCK "FVs_o/p"   // DB6
{ S7_Optimized_Access := 'FALSE' }
VERSION : 0.1
   VAR
      FV_4 : "FV_o/c";   // Химия - 1
      FV_5 : "FV_o/c";   // Химия - 2
      FV_1 : "FV_o/c";   // Подпитка
      FV_2 : "FV_o/c";   // Пар
      FV_3 : "FV_o/c";   // Стерил
   END_VAR
BEGIN
END_DATA_BLOCK

DATA_BLOCK "ЗОНЫ_Параметры"   // DB15
{ S7_Optimized_Access := 'FALSE' }
VERSION : 0.1
   VAR
      Zone_1 : "Zone_Pararm";
      Zone_2 : "Zone_Pararm";
      Zone_3 : "Zone_Pararm";
      Zone_4 : "Zone_Pararm";
      Zone_5 : "Zone_Pararm";
      Zone_6 : "Zone_Pararm";
      Zone_7 : "Zone_Pararm";
      Zone_8 : "Zone_Pararm";
      Zone_9 : "Zone_Pararm";
      Zone_10 : "Zone_Pararm";
   END_VAR
BEGIN
   Zone_1.rSet := 30.0;
   Zone_2.rTemp := 0.0;
   Zone_5.rTemp := 0.0;
   Zone_1.rDeltaDown := 3.0;
   Zone_2.rDeltaDown := 3.0;
   Zone_3.rDeltaDown := 3.0;
   Zone_5.rDeltaDown := 3.0;
   Zone_2.rSet := 60.0;
   Zone_5.rSet := 55.0;
   Zone_3.bPriority := true;
   Zone_3.rSet := 65.0;
   Zone_4.rSet := 60.0;
   Zone_6.rSet := 40.0;
   Zone_8.rSet := 10.0;
   Zone_9.rSet := 5.0;
   Zone_10.rSet := 1.0;
END_DATA_BLOCK

DATA_BLOCK "FVs_Regul"   // DB24
{ S7_Optimized_Access := 'FALSE' }
VERSION : 0.1
   VAR
      FV_Regul_1 : "FV_regul";   // Зона - 1
      FV_Regul_2 : "FV_regul";   // Зона - 2
      FV_Regul_3 : "FV_regul";   // Зона 3
      FV_Regul_4 : "FV_regul";   // Зона 4
      FV_Regul_5 : "FV_regul";   // Зона 5
      FV_Regul_6 : "FV_regul";   // Зона 6
      FV_Regul_7 : "FV_regul";   // Зона 10 - Холод
      FV_Regul_8 : "FV_regul";   // Зона 3 - охлаждение (Аварийное)
      FV_Regul_9 : "FV_regul";   // Зона 4 - охлаждение (Аварийное)
      FV_Regul_10 : "FV_regul";   // Зона 5 - охлаждение (аварийное)
      FV_Regul_11 : "FV_regul";   // Зона 6 - Охлаждение (Аварийное)
      FV_Regul_12 : "FV_regul";   // Зона 7 Охлаждение (Аварийное)
   END_VAR
BEGIN
END_DATA_BLOCK

DATA_BLOCK "Pumps"   // DB30
{ S7_Optimized_Access := 'FALSE' }
VERSION : 0.1
   VAR
      Pump_1 : "tipe_Pumps";
      Pump_2 : "tipe_Pumps";
      Pump_3 : "tipe_Pumps";
      Pump_4 : "tipe_Pumps";
      Pump_5 : "tipe_Pumps";
      Pump_6 : "tipe_Pumps";
      Pump_7 : "tipe_Pumps";
      Pump_8 : "tipe_Pumps";
      Pump_9 : "tipe_Pumps";
      Pump_10 : "tipe_Pumps";
   END_VAR
BEGIN
   Pump_1.bIn_AutomatState := true;
   Pump_2.bIn_AutomatState := true;
   Pump_3.bIn_AutomatState := true;
   Pump_4.bIn_AutomatState := true;
   Pump_5.bIn_AutomatState := true;
   Pump_6.bIn_AutomatState := true;
   Pump_7.bIn_AutomatState := true;
   Pump_8.bIn_AutomatState := true;
   Pump_9.bIn_AutomatState := true;
   Pump_10.bIn_AutomatState := true;
END_DATA_BLOCK

DATA_BLOCK "DI"   // DB43
{ S7_Optimized_Access := 'FALSE' }
VERSION : 0.1
   VAR
      DI_0 : "Tipe_DI";
      DI_1 : "Tipe_DI";
      DI_2 : "Tipe_DI";
      DI_3 : "Tipe_DI";
      DI_4 : "Tipe_DI";
      DI_5 : "Tipe_DI";
      DI_6 : "Tipe_DI";
      DI_7 : "Tipe_DI";
      DI_8 : "Tipe_DI";
      DI_9 : "Tipe_DI";
      DI_10 : "Tipe_DI";
      DI_11 : "Tipe_DI";
      DI_12 : "Tipe_DI";
      DI_13 : "Tipe_DI";
      DI_14 : "Tipe_DI";
      DI_15 : "Tipe_DI";
      DI_16 : "Tipe_DI";
      DI_17 : "Tipe_DI";
      DI_18 : "Tipe_DI";
      DI_19 : "Tipe_DI";
      DI_20 : "Tipe_DI";
      DI_21 : "Tipe_DI";
      DI_22 : "Tipe_DI";
      DI_23 : "Tipe_DI";
   END_VAR
BEGIN
END_DATA_BLOCK

DATA_BLOCK "Conveyor"   // DB82
{ S7_Optimized_Access := 'FALSE' }
VERSION : 0.1
   VAR
      Conveyor_1 : "Tipe_Conveyor";
      Conveyor_2 : "Tipe_Conveyor";
      Conveyor_3 : "Tipe_Conveyor";
      Conveyor_4 : "Tipe_Conveyor";
   END_VAR
BEGIN
   Conveyor_1.rManualSpeed := 0.0;
   Conveyor_1.rAutoSpeed := 70.0;
   Conveyor_2.rAutoSpeed := 50.0;
   Conveyor_3.rAutoSpeed := 60.0;
   Conveyor_4.rAutoSpeed := 70.0;
   Conveyor_1.bIn_AutomatState := true;
   Conveyor_2.bIn_AutomatState := true;
   Conveyor_3.bIn_AutomatState := true;
   Conveyor_4.bIn_AutomatState := true;
END_DATA_BLOCK

DATA_BLOCK "Vent"   // DB83
{ S7_Optimized_Access := 'FALSE' }
VERSION : 0.1
   VAR
      Vent_1 : "tipe_Pumps";   // Вентилятор обдува
   END_VAR
BEGIN
   Vent_1.bIn_AutomatState := true;
END_DATA_BLOCK

DATA_BLOCK "Filling_BacLevel"   // DB85
{ S7_Optimized_Access := 'FALSE' }
VERSION : 0.1
   VAR
      "1" : "Tipe_Filling_Bac";   // 1 бак
   END_VAR
BEGIN
   "1".diTimeCloseValve := 5;
END_DATA_BLOCK

DATA_BLOCK "Alarms"   // DB87
{ S7_Optimized_Access := 'FALSE' }
VERSION : 0.1
   VAR
      Ai_Alarm : Array[1..7] of Struct   // Аварии датчиков аналоговых
         ALARM : Bool;
         RESET : Bool;
      END_STRUCT;
      Pump_Alarm : Array[1..10] of Struct   // Аварии насосов
         ALARM : Bool;
         RESET : Bool;
      END_STRUCT;
      Conveyor_Alarm : Array[1..4] of Struct   // Аварии конвейеров
         ALARM : Bool;
         RESET : Bool;
      END_STRUCT;
      Vent_Alarm : Struct   // Авария вентиляторов
         Vent_Alarm_1 : Bool;
         RESET : Bool;
      END_STRUCT;
      Avtomat_Off : Array[1..11] of Struct   // Контроль состояния вкл мотор автоматов
         ALARM : Bool;
      END_STRUCT;
      FV_Alarm : Array[1..7] of Struct   // Авария клапанов
         ALARM : Bool;
         RESET : Bool;
      END_STRUCT;
      "xE-Stop_1" : Bool;   // Авария по кнопке 1
      "xE-Stop_2" : Bool;   // Авария по кнопке 2
      "xE-Stop_3" : Bool;   // Авария по кнопке 3
      xVoltRele : Bool;   // Авария реле контроля фаз
      xSensorConveyorZator_1 : Bool;   // Авария затор на конвейере - 1
      xSensorConveyorZator_2 : Bool;   // Авария затор на конвейере - 2
      xLongPauseConv : Bool;   // Авария, долгое ожидание выхода конвейера из паузы
      xLongWaitZoneOk : Bool;   // Ааврия, долгий выход на уставки
   END_VAR
BEGIN
END_DATA_BLOCK

DATA_BLOCK "AI_DB"   // DB90
{ S7_Optimized_Access := 'FALSE' }
VERSION : 0.1
   VAR
      AI_1 : "Tipe_AI";   // тт-1
      AI_2 : "Tipe_AI";   // тт-1
      AI_3 : "Tipe_AI";   // тт-1
      AI_4 : "Tipe_AI";   // тт-1
      AI_5 : "Tipe_AI";   // тт-1
      AI_6 : "Tipe_AI";   // тт-1
      AI_7 : "Tipe_AI";   // тт-1
      AI_8 : "Tipe_AI";   // тт-1
      AI_9 : "Tipe_AI";   // тт-1
      AI_10 : "Tipe_AI";   // тт-1
      "AI_4-20_1" : "Tipe_AI";   // Пар
      "AI_4-20_2" : "Tipe_AI";   // Вода
      "AI_4-20_3" : "Tipe_AI";   // Гликоль
   END_VAR
BEGIN
   "AI_4-20_1".rSensor_HL := 10.0;
   "AI_4-20_2".rSensor_HL := 10.0;
   "AI_4-20_3".rSensor_HL := 10.0;
   "AI_4-20_1".bFiltr := true;
   "AI_4-20_2".bFiltr := true;
   "AI_4-20_3".bFiltr := true;
   AI_1.bFiltr := true;
   AI_2.bFiltr := true;
   AI_3.bFiltr := true;
   AI_4.bFiltr := true;
   AI_5.bFiltr := true;
END_DATA_BLOCK

DATA_BLOCK "Control_Press_DB"   // DB95
{ S7_Optimized_Access := 'FALSE' }
VERSION : 0.1
   VAR
      PressWater : "tipePress";
      PressSteam : "tipePress";
      PressGlikol : "tipePress";
   END_VAR
BEGIN
   PressWater.rSetpoint := 0.0;
   PressSteam.rSetpoint := 0.0;
   PressGlikol.rSetpoint := 0.0;
END_DATA_BLOCK

DATA_BLOCK "Зоны_Стерилизации_Парам"   // DB104
{ S7_Optimized_Access := 'FALSE' }
VERSION : 0.1
   VAR
      "Steril_Zona-1" : "Zone_Pararm";   // параметры стерилизации зона-1
      "Steril_Zona-2" : "Zone_Pararm";   // параметры стерилизации зона-2
      "Steril_Zona-3" : "Zone_Pararm";   // параметры стерилизации зона-3
      "Steril_Zona-4" : "Zone_Pararm";   // параметры стерилизации зона-4
      "Steril_Zona-5" : "Zone_Pararm";   // параметры стерилизации зона-5
      "Steril_Zona-6" : "Zone_Pararm";   // параметры стерилизации зона-6
      "Steril_Zona-7" : "Zone_Pararm";   // параметры стерилизации зона-7
      "Steril_Zona-8" : "Zone_Pararm";   // параметры стерилизации зона-7
      "Steril_Zona-9" : "Zone_Pararm";   // параметры стерилизации зона-7
      "Steril_Zona-10" : "Zone_Pararm";   // параметры стерилизации зона-7
   END_VAR
BEGIN
END_DATA_BLOCK

DATA_BLOCK "My_VarS"   // DB119
{ S7_Optimized_Access := 'FALSE' }
VERSION : 0.1
   VAR
      b_Woter_LowLevel_T1 : Bool;   // Низкий Уровень воды Танк-1
      b_Woter_UpLewel_T1 : Bool;   // Верхний Уровень воды Танк-2
   END_VAR
BEGIN
END_DATA_BLOCK

DATA_BLOCK "НасосыХимии"   // DB150
{ S7_Optimized_Access := 'FALSE' }
VERSION : 0.1
   VAR
      Pump_Him_1 : "tipePumpHim";
      Pump_Him_2 : "tipePumpHim";
   END_VAR
BEGIN
END_DATA_BLOCK

DATA_BLOCK "Зоны_Баня_Парам"   // DB155
{ S7_Optimized_Access := 'FALSE' }
VERSION : 0.1
   VAR
      "Banya_Zona-4" : "Zone_Pararm";   // параметры стерилизации зона-4
      "Banya_Zona-5" : "Zone_Pararm";   // параметры стерилизации зона-5
      "Banya_Zona-6" : "Zone_Pararm";   // параметры стерилизации зона-6
   END_VAR
BEGIN
END_DATA_BLOCK

DATA_BLOCK "Param_PID"   // DB158
{ S7_Optimized_Access := 'FALSE' }
VERSION : 0.1
   VAR
      k_PID_Zona1 : "Коэф ПИД";   // ПИД - ЗОна 1
      k_PID_Zona2 : "Коэф ПИД";   // ПИД - зона 2
      k_PID_Zona3 : "Коэф ПИД";   // ПИД - ЗОна 3
      k_PID_Zona4 : "Коэф ПИД";   // ПИД - зона 4
      k_PID_Zona5 : "Коэф ПИД";   // ПИД - зона 5
      k_PID_Zona6 : "Коэф ПИД";   // ПИД - зона 6
      k_PID_Zona10 : "Коэф ПИД";   // ПИД - ЗОна 10 - охлаждение
      k_PID_Zona3_Охл : "Коэф ПИД";   // ПИД - ЗОна 3 - охлаждение - аварийный
      k_PID_Zona4_Охл : "Коэф ПИД";   // ПИД - ЗОна 4 - охлаждение - аварийный
      k_PID_Zona5_Охл : "Коэф ПИД";   // ПИД - ЗОна 5 - охлаждение - аварийный
      k_PID_Zona6_Охл : "Коэф ПИД";   // ПИД - ЗОна 6 - охлаждение - аварийный
      k_PID_Zona7_Охл : "Коэф ПИД";   // ПИД - ЗОна 7 - охлаждение - аварийный
   END_VAR
BEGIN
   k_PID_Zona1.Gain := 1;
   k_PID_Zona1.I := 20;
   k_PID_Zona2.Gain := 1;
   k_PID_Zona2.I := 20;
   k_PID_Zona3.Gain := 1;
   k_PID_Zona3.I := 20;
   k_PID_Zona4.Gain := 1;
   k_PID_Zona4.I := 20;
   k_PID_Zona5.Gain := 1;
   k_PID_Zona5.I := 20;
   k_PID_Zona6.Gain := 1;
   k_PID_Zona6.I := 20;
   k_PID_Zona10.Gain := 1;
   k_PID_Zona10.I := 20;
   k_PID_Zona3_Охл.Gain := 1;
   k_PID_Zona3_Охл.I := 20;
   k_PID_Zona4_Охл.Gain := 1;
   k_PID_Zona4_Охл.I := 20;
   k_PID_Zona5_Охл.Gain := 1;
   k_PID_Zona5_Охл.I := 20;
   k_PID_Zona6_Охл.Gain := 1;
   k_PID_Zona6_Охл.I := 20;
   k_PID_Zona7_Охл.Gain := 1;
   k_PID_Zona7_Охл.I := 20;
END_DATA_BLOCK

DATA_BLOCK "Param_Speed_Conv"   // DB166
{ S7_Optimized_Access := 'TRUE' }
VERSION : 0.1
   VAR RETAIN
      rLangh_Pulse : Real := 0.001;   // м, Расстояние пройденное за один импульс
      rCoef_AlfaFilter : Real := 0.1;   // Плавность изменения занчений
      tMax_Pause : DInt := 3000;   // мс, Считать остановкой если нет импульсов
      tMinPulse : DInt := 5;   // мс, Антидребезг
   END_VAR
BEGIN
END_DATA_BLOCK

DATA_BLOCK "DB_PE_Calc_V1"   // DB171
{ S7_Optimized_Access := 'FALSE' }
VERSION : 0.1
   VAR
      HMI_PE : "PE_Param";
   END_VAR
BEGIN
   HMI_PE.rПЕ_Задан := 65.0;
   HMI_PE.rДлина_Конв := 2.1;
   HMI_PE.rТемп_Макс := 100.0;
   HMI_PE."rСкоростьКонв_м/мин" := 0.24;
   HMI_PE.diВремяПростоя := 900000;
END_DATA_BLOCK

DATA_BLOCK "DB_ParamADDr_RS485"   // DB198
{ S7_Optimized_Access := 'FALSE' }
VERSION : 0.1
   VAR
      sParam_RS485 : Array[1..12] of Struct
         MB_ARRD : Int;   // Адрес устройства
         MB_MODE : Int;   // 0 - чтение 1 - запись
         MB_Registr : UInt;   // Регистр
         MB_LEN : Int;   // Кол-во регистров чтения за раз
         MB_Value : UInt;   // Значение для регистра
      END_STRUCT;
   END_VAR
BEGIN
   sParam_RS485[1].MB_ARRD := 1;
   sParam_RS485[2].MB_ARRD := 2;
   sParam_RS485[3].MB_ARRD := 3;
   sParam_RS485[1].MB_MODE := 1;
   sParam_RS485[2].MB_MODE := 1;
   sParam_RS485[1].MB_Registr := 40031;
   sParam_RS485[1].MB_LEN := 1;
   sParam_RS485[2].MB_Registr := 40031;
   sParam_RS485[2].MB_LEN := 1;
   sParam_RS485[3].MB_MODE := 1;
   sParam_RS485[3].MB_Registr := 40031;
   sParam_RS485[3].MB_LEN := 1;
   sParam_RS485[4].MB_ARRD := 4;
   sParam_RS485[4].MB_MODE := 1;
   sParam_RS485[4].MB_Registr := 40031;
   sParam_RS485[4].MB_LEN := 1;
   sParam_RS485[5].MB_ARRD := 5;
   sParam_RS485[5].MB_MODE := 1;
   sParam_RS485[5].MB_Registr := 40031;
   sParam_RS485[5].MB_LEN := 1;
   sParam_RS485[6].MB_ARRD := 6;
   sParam_RS485[6].MB_MODE := 1;
   sParam_RS485[6].MB_Registr := 40031;
   sParam_RS485[6].MB_LEN := 1;
   sParam_RS485[7].MB_ARRD := 7;
   sParam_RS485[7].MB_MODE := 1;
   sParam_RS485[7].MB_Registr := 40031;
   sParam_RS485[7].MB_LEN := 1;
   sParam_RS485[8].MB_ARRD := 8;
   sParam_RS485[8].MB_MODE := 1;
   sParam_RS485[8].MB_Registr := 40031;
   sParam_RS485[8].MB_LEN := 1;
   sParam_RS485[9].MB_ARRD := 9;
   sParam_RS485[9].MB_MODE := 1;
   sParam_RS485[9].MB_Registr := 40031;
   sParam_RS485[9].MB_LEN := 1;
   sParam_RS485[10].MB_ARRD := 10;
   sParam_RS485[10].MB_MODE := 1;
   sParam_RS485[10].MB_Registr := 40031;
   sParam_RS485[10].MB_LEN := 1;
   sParam_RS485[11].MB_ARRD := 11;
   sParam_RS485[11].MB_MODE := 1;
   sParam_RS485[11].MB_Registr := 40031;
   sParam_RS485[11].MB_LEN := 1;
   sParam_RS485[12].MB_ARRD := 12;
   sParam_RS485[12].MB_MODE := 1;
   sParam_RS485[12].MB_Registr := 40031;
   sParam_RS485[12].MB_LEN := 1;
END_DATA_BLOCK

// folder: Use VARs to HMI/DB_PE_V2

DATA_BLOCK "DB_Config"   // DB172
{ S7_Optimized_Access := 'FALSE' }
VERSION : 0.1
   VAR
      c_BaseTemp : Real := 60.0;   // Базовая температура пастеризации
      c_Z_Value : Real := 10.0;   // Z-значение
      c_Factor : Real := 1.393;   // Основание степени
      c_MaxTempDev : Real := 2.0;   // Доп. отклонение T воды (°C)
      c_StopLimit_Short : Time := t#2m;   // Лимит короткого простоя
      c_StopLimit_Long : Time := t#5m;   // Лимит длинного простоя
      c_TunnelPositions : Int := 100;   // Кол-во виртуальных позиций
      c_PosLength : Real := 0.12;   // Длина 1 позиции (м)
   END_VAR
BEGIN
END_DATA_BLOCK

DATA_BLOCK "DB_Recipe"   // DB173
{ S7_Optimized_Access := 'FALSE' }
VERSION : 0.1
   VAR
      Recipe_PE : "Recipe";
   END_VAR
BEGIN
END_DATA_BLOCK

DATA_BLOCK "DB_Status"   // DB174
{ S7_Optimized_Access := 'FALSE' }
VERSION : 0.1
   VAR
      Status_PE : "Status_V2";
   END_VAR
BEGIN
END_DATA_BLOCK

DATA_BLOCK "DB_Alarm"   // DB175
{ S7_Optimized_Access := 'FALSE' }
VERSION : 0.1
   VAR
      Alarm_PE : "Alarm";
   END_VAR
BEGIN
END_DATA_BLOCK

DATA_BLOCK "DB_StopMgr"   // DB176
{ S7_Optimized_Access := 'FALSE' }
VERSION : 0.1
   VAR
      StopMgr_PE : "StopMgr";
   END_VAR
BEGIN
END_DATA_BLOCK

DATA_BLOCK "DB_Tunnel"   // DB177
{ S7_Optimized_Access := 'FALSE' }
VERSION : 0.1
   VAR
      Tunel_Virt_Pe : Array[1..100] of "ProductPosition";
   END_VAR
BEGIN
END_DATA_BLOCK

DATA_BLOCK "DB_TempWater_Fact"   // DB179
{ S7_Optimized_Access := 'TRUE' }
VERSION : 0.1
BEGIN
END_DATA_BLOCK

// folder: Use VARs to HMI/DB_PE_V3

DATA_BLOCK "DB_StopMGR_V3"   // DB182
{ S7_Optimized_Access := 'TRUE' }
VERSION : 0.1
   VAR
      StopMGR_PE_V3 : "StopMgr";
   END_VAR
BEGIN
END_DATA_BLOCK

DATA_BLOCK "DB_Status_V3"   // DB183
{ S7_Optimized_Access := 'FALSE' }
VERSION : 0.1
   VAR
      Status_V3_PE : "Status_V3";
   END_VAR
BEGIN
END_DATA_BLOCK

DATA_BLOCK "DB_Alarm_V3"   // DB184
{ S7_Optimized_Access := 'FALSE' }
VERSION : 0.1
   VAR
      Alarm_V3_Pe : "Alarm";
   END_VAR
BEGIN
END_DATA_BLOCK

DATA_BLOCK "Temp_ZONE_Arrey"   // DB185
{ S7_Optimized_Access := 'FALSE' }
VERSION : 0.1
   VAR
      TempZone : Array[1..9] of Real;
   END_VAR
BEGIN
END_DATA_BLOCK

DATA_BLOCK "DB_Param_Calc_PE"   // DB186
{ S7_Optimized_Access := 'FALSE' }
VERSION : 0.1
   VAR
      cR_BaseTemp : Real := 60.0;   // Базовая температура пастеризации
      cR_Z_Value : Real := 10.0;   // Z-значение - 10
      cR_Factor : Real := 1.393;   // Основание степени, 1.393
      cR_K_Coeff : Real := 7.0;   // Коэффициент теплопередачи (1/мин)
      cR_PU_Target_Min : Real;   // Минимально допустимые ПЕ
      cR_PU_Target_Max : Real;   // Максимально допустимые ПЕ
      cR_TempProd_Inlet : Real := 2.0;   // Температура продукта на входе (°C)
      cR_MaxTempDev : Real := 2.0;   // Доп. отклонение T воды (°C)
      cR_StopLimit_Short : Real := 2.0;   // Лимит короткого простоя, мин
      cR_StopLimit_Long : Real := 5.0;   // Лимит длинного простоя, мин
   END_VAR
BEGIN
END_DATA_BLOCK

DATA_BLOCK "DB_Config_Zones"   // DB191
{ S7_Optimized_Access := 'FALSE' }
VERSION : 0.1
   VAR
      ZoneConfig : Array[1..9] of "Zone_Config_V3";
   END_VAR
BEGIN
   ZoneConfig[1].Length := 1.2;
   ZoneConfig[2].Length := 1.2;
   ZoneConfig[3].Length := 1.2;
   ZoneConfig[4].Length := 1.2;
   ZoneConfig[5].Length := 1.2;
   ZoneConfig[6].Length := 1.2;
   ZoneConfig[7].Length := 1.2;
   ZoneConfig[8].Length := 1.2;
   ZoneConfig[9].Length := 1.2;
END_DATA_BLOCK

// folder: Use VARs to HMI/DB_PE_V3/PE_Расчет

DATA_BLOCK "Temp_ZONE_Для Расчетной ПЕ"   // DB187
{ S7_Optimized_Access := 'FALSE' }
VERSION : 0.1
   VAR
      TempZone : Array[1..9] of Real;
   END_VAR
BEGIN
END_DATA_BLOCK

DATA_BLOCK "DB_StopMGR__Для Расчетной ПЕ"   // DB188
{ S7_Optimized_Access := 'TRUE' }
VERSION : 0.1
   VAR
      StopMGR_PE_V3 : "StopMgr";
   END_VAR
BEGIN
END_DATA_BLOCK

DATA_BLOCK "DB_Status_Для Расчетной ПЕ"   // DB189
{ S7_Optimized_Access := 'FALSE' }
VERSION : 0.1
   VAR
      Status_V3_PE : "Status_V3";
   END_VAR
BEGIN
END_DATA_BLOCK

DATA_BLOCK "DB_Alarm_Для Расчетной ПЕ"   // DB190
{ S7_Optimized_Access := 'FALSE' }
VERSION : 0.1
   VAR
      Alarm_V3_Pe : "Alarm";
   END_VAR
BEGIN
END_DATA_BLOCK

// folder: Зоны/DB_Zone

DATA_BLOCK "FB_Zone_Control_1_DB"   // DB12
{ S7_Optimized_Access := 'FALSE' }
VERSION : 0.1
// stored: InstanceOfName FB_Zone_Control
"FB_Zone_Control"
BEGIN
END_DATA_BLOCK

DATA_BLOCK "FB_Zone_Control_2_DB"   // DB13
{ S7_Optimized_Access := 'FALSE' }
VERSION : 0.1
// stored: InstanceOfName FB_Zone_Control
"FB_Zone_Control"
BEGIN
END_DATA_BLOCK

DATA_BLOCK "FB_Zone_Control_3_DB"   // DB14
{ S7_Optimized_Access := 'FALSE' }
VERSION : 0.1
// stored: InstanceOfName FB_Zone_Control
"FB_Zone_Control"
BEGIN
END_DATA_BLOCK

DATA_BLOCK "FB_Zone_Control_4_DB"   // DB16
{ S7_Optimized_Access := 'FALSE' }
VERSION : 0.1
// stored: InstanceOfName FB_Zone_Control
"FB_Zone_Control"
BEGIN
END_DATA_BLOCK

DATA_BLOCK "FB_Zone_Control_5_DB"   // DB17
{ S7_Optimized_Access := 'FALSE' }
VERSION : 0.1
// stored: InstanceOfName FB_Zone_Control
"FB_Zone_Control"
BEGIN
END_DATA_BLOCK

DATA_BLOCK "FB_Zone_Control_7_DB"   // DB94
{ S7_Optimized_Access := 'FALSE' }
VERSION : 0.1
// stored: InstanceOfName FB_Zone_Control
"FB_Zone_Control"
BEGIN
END_DATA_BLOCK

DATA_BLOCK "FB_Zone_Control_6_DB"   // DB114
{ S7_Optimized_Access := 'FALSE' }
VERSION : 0.1
// stored: InstanceOfName FB_Zone_Control
"FB_Zone_Control"
BEGIN
END_DATA_BLOCK

DATA_BLOCK "FB_Zone_4_Control_Banya_DB"   // DB120
{ S7_Optimized_Access := 'FALSE' }
VERSION : 0.1
// stored: InstanceOfName FB_Zone_Control_Steriliz
"FB_Zone_Control_Steriliz"
BEGIN
END_DATA_BLOCK

DATA_BLOCK "FB_Zone_Control_8_DB"   // DB131
{ S7_Optimized_Access := 'FALSE' }
VERSION : 0.1
// stored: InstanceOfName FB_Zone_Control
"FB_Zone_Control"
BEGIN
END_DATA_BLOCK

DATA_BLOCK "FB_Zone_Control_9_DB"   // DB132
{ S7_Optimized_Access := 'FALSE' }
VERSION : 0.1
// stored: InstanceOfName FB_Zone_Control
"FB_Zone_Control"
BEGIN
END_DATA_BLOCK

DATA_BLOCK "FB_Zone_Control_10_DB"   // DB133
{ S7_Optimized_Access := 'FALSE' }
VERSION : 0.1
// stored: InstanceOfName FB_Zone_Control
"FB_Zone_Control"
BEGIN
END_DATA_BLOCK

DATA_BLOCK "FB_Zone_5_Control_Banya_DB"   // DB153
{ S7_Optimized_Access := 'FALSE' }
VERSION : 0.1
// stored: InstanceOfName FB_Zone_Control_Steriliz
"FB_Zone_Control_Steriliz"
BEGIN
END_DATA_BLOCK

DATA_BLOCK "FB_Zone_6_Control_Banya_DB"   // DB154
{ S7_Optimized_Access := 'FALSE' }
VERSION : 0.1
// stored: InstanceOfName FB_Zone_Control_Steriliz
"FB_Zone_Control_Steriliz"
BEGIN
END_DATA_BLOCK

// folder: Зоны/Стерилизация

DATA_BLOCK "FB_Zone_1_Control_Steriliz_DB"   // DB105
{ S7_Optimized_Access := 'FALSE' }
VERSION : 0.1
// stored: InstanceOfName FB_Zone_Control_Steriliz
"FB_Zone_Control_Steriliz"
BEGIN
END_DATA_BLOCK

DATA_BLOCK "FB_Zone_2_Control_Стерилизация_DB"   // DB106
{ S7_Optimized_Access := 'FALSE' }
VERSION : 0.1
// stored: InstanceOfName FB_Zone_Control_Steriliz
"FB_Zone_Control_Steriliz"
BEGIN
END_DATA_BLOCK

DATA_BLOCK "FB_Zone_3_Control_Стерилизация_DB"   // DB107
{ S7_Optimized_Access := 'FALSE' }
VERSION : 0.1
// stored: InstanceOfName FB_Zone_Control_Steriliz
"FB_Zone_Control_Steriliz"
BEGIN
END_DATA_BLOCK

DATA_BLOCK "FB_Zone_4_Control_Стерилизация_DB"   // DB108
{ S7_Optimized_Access := 'FALSE' }
VERSION : 0.1
// stored: InstanceOfName FB_Zone_Control_Steriliz
"FB_Zone_Control_Steriliz"
BEGIN
END_DATA_BLOCK

DATA_BLOCK "FB_Zone_5_Control_Стерилизация_DB"   // DB109
{ S7_Optimized_Access := 'FALSE' }
VERSION : 0.1
// stored: InstanceOfName FB_Zone_Control_Steriliz
"FB_Zone_Control_Steriliz"
BEGIN
END_DATA_BLOCK

DATA_BLOCK "FB_Zone_6_Control_Стерилизация_DB"   // DB110
{ S7_Optimized_Access := 'FALSE' }
VERSION : 0.1
// stored: InstanceOfName FB_Zone_Control_Steriliz
"FB_Zone_Control_Steriliz"
BEGIN
END_DATA_BLOCK

DATA_BLOCK "FB_Zone_7_Control_Стерилизация_DB"   // DB111
{ S7_Optimized_Access := 'FALSE' }
VERSION : 0.1
// stored: InstanceOfName FB_Zone_Control_Steriliz
"FB_Zone_Control_Steriliz"
BEGIN
END_DATA_BLOCK

DATA_BLOCK "FB_Zone_8_Control_Стерилизация_DB"   // DB134
{ S7_Optimized_Access := 'FALSE' }
VERSION : 0.1
// stored: InstanceOfName FB_Zone_Control_Steriliz
"FB_Zone_Control_Steriliz"
BEGIN
END_DATA_BLOCK

DATA_BLOCK "FB_Zone_9_Control_Стерилизация_DB"   // DB135
{ S7_Optimized_Access := 'FALSE' }
VERSION : 0.1
// stored: InstanceOfName FB_Zone_Control_Steriliz
"FB_Zone_Control_Steriliz"
BEGIN
END_DATA_BLOCK

DATA_BLOCK "FB_Zone_10_Control_Стерилизация_DB"   // DB136
{ S7_Optimized_Access := 'FALSE' }
VERSION : 0.1
// stored: InstanceOfName FB_Zone_Control_Steriliz
"FB_Zone_Control_Steriliz"
BEGIN
END_DATA_BLOCK

// folder: Клапана/FV_o/C/FV_DB

DATA_BLOCK "FV_1"   // DB4
{ S7_Optimized_Access := 'FALSE' }
VERSION : 0.1
// stored: InstanceOfName Valve(c/o)
"Valve(c/o)"
BEGIN
END_DATA_BLOCK

DATA_BLOCK "FV_2"   // DB9
{ S7_Optimized_Access := 'FALSE' }
VERSION : 0.1
// stored: InstanceOfName Valve(c/o)
"Valve(c/o)"
BEGIN
END_DATA_BLOCK

DATA_BLOCK "FV_3"   // DB10
{ S7_Optimized_Access := 'FALSE' }
VERSION : 0.1
// stored: InstanceOfName Valve(c/o)
"Valve(c/o)"
BEGIN
END_DATA_BLOCK

DATA_BLOCK "FV_4_НасХимия_1"   // DB147
{ S7_Optimized_Access := 'FALSE' }
VERSION : 0.1
// stored: InstanceOfName Valve(c/o)
"Valve(c/o)"
BEGIN
END_DATA_BLOCK

DATA_BLOCK "FV_5"   // DB148
{ S7_Optimized_Access := 'FALSE' }
VERSION : 0.1
// stored: InstanceOfName Valve(c/o)
"Valve(c/o)"
BEGIN
END_DATA_BLOCK

// folder: Клапана/FV_regul/DB

DATA_BLOCK "FV_Regul_1_DB"   // DB20
{ S7_Optimized_Access := 'FALSE' }
VERSION : 0.1
// stored: InstanceOfName Valve(regul)
"Valve(regul)"
BEGIN
END_DATA_BLOCK

DATA_BLOCK "FV_Regul_2_DB"   // DB21
{ S7_Optimized_Access := 'FALSE' }
VERSION : 0.1
// stored: InstanceOfName Valve(regul)
"Valve(regul)"
BEGIN
END_DATA_BLOCK

DATA_BLOCK "FV_Regul_3_DB"   // DB22
{ S7_Optimized_Access := 'FALSE' }
VERSION : 0.1
// stored: InstanceOfName Valve(regul)
"Valve(regul)"
BEGIN
END_DATA_BLOCK

DATA_BLOCK "FV_Regul_4_DB"   // DB23
{ S7_Optimized_Access := 'FALSE' }
VERSION : 0.1
// stored: InstanceOfName Valve(regul)
"Valve(regul)"
BEGIN
END_DATA_BLOCK

DATA_BLOCK "FV_Regul_5_DB"   // DB37
{ S7_Optimized_Access := 'FALSE' }
VERSION : 0.1
// stored: InstanceOfName Valve(regul)
"Valve(regul)"
BEGIN
END_DATA_BLOCK

DATA_BLOCK "FV_Regul_6_DB"   // DB140
{ S7_Optimized_Access := 'FALSE' }
VERSION : 0.1
// stored: InstanceOfName Valve(regul)
"Valve(regul)"
BEGIN
END_DATA_BLOCK

DATA_BLOCK "FV_Regul_7_DB"   // DB141
{ S7_Optimized_Access := 'FALSE' }
VERSION : 0.1
// stored: InstanceOfName Valve(regul)
"Valve(regul)"
BEGIN
END_DATA_BLOCK

DATA_BLOCK "FV_Regul_9_DB"   // DB142
{ S7_Optimized_Access := 'FALSE' }
VERSION : 0.1
// stored: InstanceOfName Valve(regul)
"Valve(regul)"
BEGIN
END_DATA_BLOCK

DATA_BLOCK "FV_Regul_10_DB"   // DB143
{ S7_Optimized_Access := 'FALSE' }
VERSION : 0.1
// stored: InstanceOfName Valve(regul)
"Valve(regul)"
BEGIN
END_DATA_BLOCK

DATA_BLOCK "FV_Regul_11_DB"   // DB144
{ S7_Optimized_Access := 'FALSE' }
VERSION : 0.1
// stored: InstanceOfName Valve(regul)
"Valve(regul)"
BEGIN
END_DATA_BLOCK

DATA_BLOCK "FV_Regul_12_DB"   // DB145
{ S7_Optimized_Access := 'FALSE' }
VERSION : 0.1
// stored: InstanceOfName Valve(regul)
"Valve(regul)"
BEGIN
END_DATA_BLOCK

DATA_BLOCK "FV_Regul_8_DB"   // DB146
{ S7_Optimized_Access := 'FALSE' }
VERSION : 0.1
// stored: InstanceOfName Valve(regul)
"Valve(regul)"
BEGIN
END_DATA_BLOCK

// folder: Конвейера/DB

DATA_BLOCK "Конвейер_1_DB"   // DB78
{ S7_Optimized_Access := 'FALSE' }
VERSION : 0.1
// stored: InstanceOfName Pump
"Pump"
BEGIN
END_DATA_BLOCK

DATA_BLOCK "Конвейер_2_DB"   // DB79
{ S7_Optimized_Access := 'FALSE' }
VERSION : 0.1
// stored: InstanceOfName Pump
"Pump"
BEGIN
END_DATA_BLOCK

DATA_BLOCK "Конвейер_3_DB"   // DB80
{ S7_Optimized_Access := 'FALSE' }
VERSION : 0.1
// stored: InstanceOfName Pump
"Pump"
BEGIN
END_DATA_BLOCK

// folder: Насосы/DB

DATA_BLOCK "Pump_6_DB"   // DB5
{ S7_Optimized_Access := 'FALSE' }
VERSION : 0.1
// stored: InstanceOfName Pump
"Pump"
BEGIN
END_DATA_BLOCK

DATA_BLOCK "Pump_7_DB"   // DB7
{ S7_Optimized_Access := 'FALSE' }
VERSION : 0.1
// stored: InstanceOfName Pump
"Pump"
BEGIN
END_DATA_BLOCK

DATA_BLOCK "Pump_1_DB"   // DB25
{ S7_Optimized_Access := 'FALSE' }
VERSION : 0.1
// stored: InstanceOfName Pump
"Pump"
BEGIN
END_DATA_BLOCK

DATA_BLOCK "Pump_2_DB"   // DB26
{ S7_Optimized_Access := 'FALSE' }
VERSION : 0.1
// stored: InstanceOfName Pump
"Pump"
BEGIN
END_DATA_BLOCK

DATA_BLOCK "Pump_5_DB"   // DB27
{ S7_Optimized_Access := 'FALSE' }
VERSION : 0.1
// stored: InstanceOfName Pump
"Pump"
BEGIN
END_DATA_BLOCK

DATA_BLOCK "Pump_4_DB"   // DB28
{ S7_Optimized_Access := 'FALSE' }
VERSION : 0.1
// stored: InstanceOfName Pump
"Pump"
BEGIN
END_DATA_BLOCK

DATA_BLOCK "Pump_3_DB"   // DB29
{ S7_Optimized_Access := 'FALSE' }
VERSION : 0.1
// stored: InstanceOfName Pump
"Pump"
BEGIN
END_DATA_BLOCK

DATA_BLOCK "Pump_8_DB"   // DB137
{ S7_Optimized_Access := 'FALSE' }
VERSION : 0.1
// stored: InstanceOfName Pump
"Pump"
BEGIN
END_DATA_BLOCK

DATA_BLOCK "Pump_9_DB"   // DB138
{ S7_Optimized_Access := 'FALSE' }
VERSION : 0.1
// stored: InstanceOfName Pump
"Pump"
BEGIN
END_DATA_BLOCK

DATA_BLOCK "Pump_10_DB"   // DB139
{ S7_Optimized_Access := 'FALSE' }
VERSION : 0.1
// stored: InstanceOfName Pump
"Pump"
BEGIN
END_DATA_BLOCK

// folder: Насосы/Химия

DATA_BLOCK "Насос химии_1DB"   // DB149
{ S7_Optimized_Access := 'TRUE' }
VERSION : 0.1
// stored: InstanceOfName Насос химии
"Насос химии"
BEGIN
END_DATA_BLOCK

DATA_BLOCK "Насос химии_2DB"   // DB151
{ S7_Optimized_Access := 'TRUE' }
VERSION : 0.1
// stored: InstanceOfName Насос химии
"Насос химии"
BEGIN
END_DATA_BLOCK

// folder: (top level)

FUNCTION_BLOCK "FB_Расчет скорости по импульсам"   // FB30, SCL
{ S7_Optimized_Access := 'TRUE' }
VERSION : 0.1
   VAR_INPUT
      bEnable : Bool;   // TRUE = разрешить расчет, FALSE = сброс
      bSensIn : Bool;   // Дискретный сигнал с датчика (0/1)
      rLang_Pulse : Real;   // [м] Расстояние за 1 импульс (константа)
      rAlpha_Filter : Real;   // [0.0..1.0] Коэфф. сглаживания (0.1 = плавный график)
      tMax_Pause : Time;   // Таймаут остановки (если нет импульсов -> скорость 0)
      tMin_Pulse : Time;   // Мин. время импульса (фильтр дребезга/шума)
   END_VAR
   VAR_OUTPUT
      "rSpeed_m/min" : Real;   // [м/мин] Текущая скорость (отфильтрованная)
      rSpeed_raw : Real;   // [м/мин] "Сырая" скорость (без фильтра)
      bStopped : Bool;   // TRUE = конвейер остановлен (нет импульсов > tMax_Pause)
   END_VAR
   VAR
      rTrig_Sensor : "R_trig";   // Детектор переднего фронта
      tTime_Now : DTL;   // Текущая метка времени (системная)
      tTime_Last : DTL;   // Метка времени предыдущего импульса
      tPeriod : Time;   // Измеренный период между импульсами
      rPeriod_MIN : Real;   // Период в минутах (для формулы)
      rSpeed_Calc : Real;   // Промежуточный расчет
      bFirst_Pulse : Bool;   // Флаг первого импульса после включения
      iOutStatusTime : Int;   // Выход для статуса чтения текущего времени
      tWatchdog : Time;   // Текущее время для контроля остановки
   END_VAR
BEGIN
   // =====================================================================
   // Назначение: Расчет скорости конвейера методом измерения периода
   // Формула: V = L_pulse / (T_now - T_last)
   // =====================================================================


   // =================================================================
   // 1. СБРОС И ИНИЦИАЛИЗАЦИЯ
   // =================================================================
   IF NOT #bEnable THEN
       #bFirst_Pulse := TRUE;
       #bStopped := true;
       #"rSpeed_m/min" := 0.0;
       #rSpeed_raw := 0.0;
       RETURN; // Выход из блока, дальнейший код не выполняется
   END_IF;

   // =================================================================
   // 2. ДЕТЕКТИРОВАНИЕ ИМПУЛЬСА (Передний фронт)
   // =================================================================

   #rTrig_Sensor(In := #bSensIn);

   // =================================================================
   // 3. ОБРАБОТКА ПРИХОДА ИМПУЛЬСА
   // =================================================================
   IF #rTrig_Sensor.Q THEN

       // Получаем точное системное время (разрешение 1 мкс)

       #iOutStatusTime := RD_SYS_T(OUT => #tTime_Now);

       // Если это не самый первый импульс после старта - считаем скорость
       IF NOT #bFirst_Pulse THEN

           // 3.1 Измеряем период: Текущее время минус время прошлого импульса вычитаем время 
           #tPeriod := T_DIFF(IN1 := #tTime_Now, IN2 := #tTime_Last);

           // 3.2 Фильтрация шума: Игнорируем слишком короткие интервалы (вибрация, дребезг)
           IF #tPeriod >= #tMin_Pulse THEN

               // 3.3 Конвертация времени в секунды (LReal) для математики
               // переводим полуенное значение периода в тип данных Real для дальнейших вычислений времени в секундах
               #rPeriod_MIN := DINT_TO_REAL(IN := (TIME_TO_DINT(IN := #tPeriod))) / 60000.0;


               // 3.4 Расчет "сырой" скорости по формуле
               // Защита от деления на ноль уже обеспечена фильтром tMin_Pulse
               #rSpeed_raw := #rLang_Pulse / #rPeriod_MIN;

               // 3.5 Экспоненциальное сглаживание (чтобы стрелка на HMI не дергалась)
               // Y_new = Alpha * X_new + (1-Alpha) * Y_old
               #"rSpeed_m/min" := #rAlpha_Filter * #rSpeed_raw + (1.0 - #rAlpha_Filter) * #"rSpeed_m/min";

               // Флаги статуса
               #bStopped := FALSE;

           END_IF; // Конец фильтра шума

       END_IF; // Конец проверки First_Pulse

       // Запоминаем время этого импульса для следующего цикла
       #tTime_Last := #tTime_Now;
       #bFirst_Pulse := FALSE;

   END_IF; // Конец обработки фронта
END_FUNCTION_BLOCK

FUNCTION_BLOCK "Расчет ПЕ по сек"   // FB31, SCL
{ S7_Optimized_Access := 'TRUE' }
VERSION : 0.1
   VAR_INPUT
      inp_Enable : Bool;   // Разрешение расчёта
      inp_LineRun : Bool;   // Конвейер работает
      inp_Jam : Bool;   // Сигнал затора
      inp_SpeedAct : Real;   // Скорость ленты (м/мин)
      inp_TempWater : Array[1..9] of Real;   // Факт. T воды по зонам
   END_VAR
   VAR_OUTPUT
      out_Status : "Status_V2";   // Статус (DB174)
      out_Alarm : "Alarm";   // Аварии (DB175)
   END_VAR
   VAR_IN_OUT
      ino_Recipe : "Recipe";   // Ссылка на рецепт (DB173)
      ino_StopMgr : "StopMgr";   // Менеджер остановок (DB176)
      ino_Tunnel : Array[1..100] of "ProductPosition";   // Туннель (DB177)
   END_VAR
   VAR
      stat_CycleTimer : IEC_TIMER;   // Таймер 1 секунда
      stat_PU_LastOut : Real;   // ПЕ последней вышедшей бутылки
      stat_PU_Flow : Real;   // Средние ПЕ в потоке
      temp_StopDuration_Min : Real;   // Длительность простоя в минутах
      temp_CalcPositions : Bool;   // Флаг: выполнять ли расчёт движения
      temp_SourcePos : Int;   // Исходная позиция (сдвиг)
   END_VAR
   VAR_TEMP
      temp_CycleTime_Min : Real;
      temp_PosIndex : Int;
      temp_ZoneIdx : Int;   // Время цикла (мин)
      temp_TempWater : Real;   // Счётчик позиций
      temp_DeltaT : Real;   // Исходная позиция (сдвиг)
      temp_PU_Inc : Real;   // Индекс зоны
      temp_TempMax : Real;   // T воды в текущей зоне
      temp_PU_Sum : Real;   // Изменение T продукта
      temp_PosActive : Int;   // Прирост ПЕ за цикл
      temp_TempDev : Real;   // Макс. T в туннеле Сумма ПЕ для averages
      temp_DistPerSec : Real;   // М/с дист за 1 сек
      temp_PosPerSec : Real;   // Кол-во активных позиций за 1 секунду
      temp_TempHotZones : Real;   // Отклонение T воды
   END_VAR
BEGIN

       // =================================================================
       // 1. ТАЙМЕР ЦИКЛА РАСЧЁТА (1 СЕКУНДА)
       // =================================================================

       #stat_CycleTimer.TON(IN := true, PT := t#1S);


       // Если 1 секунда ещё не прошла - выход из блока
       IF NOT #stat_CycleTimer.Q THEN
           RETURN;
       END_IF;

       // Сброс таймера для следующего цикла
       #stat_CycleTimer.TON(IN := FALSE, PT := t#0s);

       // Время цикла в минутах (для формулы ПЕ)
       #temp_CycleTime_Min := 1.0 / 60.0;

       // =================================================================
       // 2. ОБРАБОТКА ОСТАНОВКИ / ЗАТОРА
       // =================================================================
       // Флаг: можно ли выполнять расчёт движения
       #temp_CalcPositions := #inp_LineRun AND NOT #inp_Jam;

       IF NOT #temp_CalcPositions THEN
           // === РЕЖИМ ПРОСТОЯ ===

           // Запуск таймера простоя
           #ino_StopMgr.Timer_Stop.TON(IN := TRUE,
                                       PT := T#100m,ET => #ino_StopMgr.Duration);

           // Преобразование времени: TIME -> DINT -> REAL -> минуты
           // TIME_TO_DINT возвращает миллисекунды как целое число
           #temp_StopDuration_Min := DINT_TO_REAL(TIME_TO_DINT(#ino_StopMgr.Duration)) / 60000.0;

           // Флаги для управления температурой и отбраковкой
           IF #temp_StopDuration_Min > 2.0 THEN  // > 2 минут
               #out_Alarm.Temp_Deviation := TRUE;  // Сигнал для снижения уставок
           END_IF;

           IF #temp_StopDuration_Min > 5.0 THEN  // > 5 минут
               #ino_StopMgr.Reject_Required := TRUE;
           END_IF;

           // Расчёт ПЕ во время простоя (горячие зоны 5-6)
           #temp_TempHotZones := (#inp_TempWater[5] + #inp_TempWater[6]) / 2.0;

           IF #temp_TempHotZones > "DB_Config".c_BaseTemp THEN
               //__________Расчет по формуле PUstop = ___________
               #ino_StopMgr.PU_Stop_Add :=
               #temp_StopDuration_Min *
               "DB_Config".c_Factor ** ((#temp_TempHotZones - "DB_Config".c_BaseTemp) / "DB_Config".c_Z_Value);
           ELSE
               #ino_StopMgr.PU_Stop_Add := 0.0;
           END_IF;

           // Пропускаем расчёт движения (код ниже выполнится только если #temp_CalcPositions = TRUE)
       ELSE
           // === РЕЖИМ РАБОТЫ ===

           // Линия работает - сброс таймера простоя
           #ino_StopMgr.Timer_Stop.TON(IN := FALSE, PT := t#0s);
           #ino_StopMgr.Duration := T#0s;
           #ino_StopMgr.PU_Stop_Add := 0.0;
           #out_Alarm.Temp_Deviation := FALSE;
       END_IF;

       // =================================================================
       // 3-7. ОСНОВНОЙ РАСЧЁТ (выполняется ТОЛЬКО если линия работает)
       // =================================================================
       IF #temp_CalcPositions THEN

           // -------------------------------------------------------------
           // !!!!!____!!!3. РАСЧЁТ ПЕРЕМЕЩЕНИЯ ПРОДУКТА (ПОЗИЦИИ) - Не прпавильный расчет - округнляет до 0 - т.к. шаг при 1 сек 0,047 шага - переделать 3 часть кода
           // -------------------------------------------------------------
           // Сколько метров проходит лента за 1 секунду
           #temp_DistPerSec := #inp_SpeedAct / 60.0; // м/сек

           // Сколько позиций проходит за 1 секунду
           // 1 позиция = c_PosLength метров (0.12 м для 12м туннеля / 100 позиций)
           #temp_PosPerSec := #temp_DistPerSec / "DB_Config".c_PosLength;

           // Ограничение минимального смещения (избегаем дребезга)
           IF #temp_PosPerSec < 0.001 THEN
               #temp_PosPerSec := 0.0;
           END_IF;

           // -------------------------------------------------------------
           // 4. СДВИГ МАССИВА ПРОДУКТА (ИМИТАЦИЯ ДВИЖЕНИЯ ЛЕНТЫ)
           // -------------------------------------------------------------
           // Сдвигаем все позиции вперёд. Позиция 100 → выход, Позиция 1 → вход
           // Идём с конца к началу, чтобы не затереть данные при копировании

           FOR #temp_PosIndex := 100 TO 2 BY -1 DO
               // Вычисляем исходную позицию с учётом скорости
               #temp_SourcePos := #temp_PosIndex - REAL_TO_INT(#temp_PosPerSec);

               IF #temp_SourcePos < 1 THEN
                   #temp_SourcePos := 1;
               END_IF;

               // Копируем данные из предыдущей позиции в текущую
               #ino_Tunnel[#temp_PosIndex].TempProduct := #ino_Tunnel[#temp_SourcePos].TempProduct;
               #ino_Tunnel[#temp_PosIndex].PU_Accumulated := #ino_Tunnel[#temp_SourcePos].PU_Accumulated;
               #ino_Tunnel[#temp_PosIndex].InTunnel := #ino_Tunnel[#temp_SourcePos].InTunnel;
               #ino_Tunnel[#temp_PosIndex].ZoneIndex := #ino_Tunnel[#temp_SourcePos].ZoneIndex;
           END_FOR;

           // -------------------------------------------------------------
           // 5. ИНИЦИАЛИЗАЦИЯ НОВОЙ ПОЗИЦИИ НА ВХОДЕ (ПОЗИЦИЯ 1)
           // -------------------------------------------------------------
           // Если продукт движется - создаём новую позицию на входе
           IF #temp_PosPerSec > 0.001 THEN
               #ino_Tunnel[1].InTunnel := TRUE;
               #ino_Tunnel[1].TempProduct := #ino_Recipe.TempProd_Inlet;
               #ino_Tunnel[1].PU_Accumulated := 0.0;
               #ino_Tunnel[1].ZoneIndex := 1;
           END_IF;

           // -------------------------------------------------------------
           // 6. РАСЧЁТ ТЕМПЕРАТУРЫ И ПЕ ДЛЯ КАЖДОЙ ПОЗИЦИИ
           // -------------------------------------------------------------
           #temp_PU_Sum := 0.0;
           #temp_TempMax := 0.0;
           #temp_PosActive := 0;

           FOR #temp_PosIndex := 1 TO 100 DO
               IF #ino_Tunnel[#temp_PosIndex].InTunnel THEN
                   #temp_PosActive := #temp_PosActive + 1;

                   // Определяем зону по позиции
                   // 100 позиций / 9 зон ≈ 11.1 позиции на зону
                   // Позиции 1-11 = зона 1, 12-22 = зона 2, и т.д.
                   #temp_ZoneIdx := (#temp_PosIndex - 1) / 12 + 1;

                   // Ограничение диапазона зон
                   IF #temp_ZoneIdx < 1 THEN
                       #temp_ZoneIdx := 1;
                   ELSIF #temp_ZoneIdx > 9 THEN
                       #temp_ZoneIdx := 9;
                   END_IF;

                   #ino_Tunnel[#temp_PosIndex].ZoneIndex := #temp_ZoneIdx;

                   // Получаем факт. температуру воды в этой зоне
                   #temp_TempWater := #inp_TempWater[#temp_ZoneIdx];

                   // === РАСЧЁТ ИЗМЕНЕНИЯ ТЕМПЕРАТУРЫ ПРОДУКТА ===
                   // Формула: T_new = T_old + (T_water - T_old) * (1 - e^(-K * dt))
                   #temp_DeltaT := (#temp_TempWater - #ino_Tunnel[#temp_PosIndex].TempProduct) *
                   (1.0 - EXP(- #ino_Recipe.K_Coeff * #temp_CycleTime_Min));

                   #ino_Tunnel[#temp_PosIndex].TempProduct :=
                   #ino_Tunnel[#temp_PosIndex].TempProduct + #temp_DeltaT;

                   // === РАСЧЁТ ПРИРОСТА ПЕ ===
                   // Только если T продукта >= 60°C (базовая температура)
                   IF #ino_Tunnel[#temp_PosIndex].TempProduct >= "DB_Config".c_BaseTemp THEN
                       #temp_PU_Inc := #temp_CycleTime_Min *
                       "DB_Config".c_Factor **
                       ((#ino_Tunnel[#temp_PosIndex].TempProduct - "DB_Config".c_BaseTemp) /
                       "DB_Config".c_Z_Value);

                       #ino_Tunnel[#temp_PosIndex].PU_Accumulated :=
                       #ino_Tunnel[#temp_PosIndex].PU_Accumulated + #temp_PU_Inc;
                   END_IF;

                   // Сбор статистики по туннелю
                   IF #ino_Tunnel[#temp_PosIndex].TempProduct > #temp_TempMax THEN
                       #temp_TempMax := #ino_Tunnel[#temp_PosIndex].TempProduct;
                   END_IF;

                   #temp_PU_Sum := #temp_PU_Sum + #ino_Tunnel[#temp_PosIndex].PU_Accumulated;
               END_IF;
           END_FOR;

           // -------------------------------------------------------------
           // 7. ОБРАБОТКА ВЫХОДА ПРОДУКТА ИЗ ТУННЕЛЯ (ПОЗИЦИЯ 100)
           // -------------------------------------------------------------
           IF #ino_Tunnel[100].InTunnel AND #temp_PosPerSec > 0.01 THEN
               // Продукт выходит из туннеля - сохраняем ПЕ для отчёта
               #stat_PU_LastOut := #ino_Tunnel[100].PU_Accumulated;

               // Проверка на недопастеризацию (ПУ ниже минимума)
               IF #stat_PU_LastOut < #ino_Recipe.PU_Target_Min THEN
                   #out_Alarm.PU_Under := TRUE;
                   #out_Alarm.Stop_Request := TRUE;
               END_IF;

               // Проверка на перепастеризацию (ПУ выше максимума)
               IF #stat_PU_LastOut > #ino_Recipe.PU_Target_Max THEN
                   #out_Alarm.PU_Over := TRUE;
                   #out_Alarm.Stop_Request := TRUE;
               END_IF;

               // Очищаем позицию после выхода продукта
               #ino_Tunnel[100].InTunnel := FALSE;
               #ino_Tunnel[100].PU_Accumulated := 0.0;
               #ino_Tunnel[100].TempProduct := 0.0;
               #ino_Tunnel[100].ZoneIndex := 0;
           END_IF;

       END_IF;  // Конец IF #temp_CalcPositions

       // =================================================================
       // 8. ЗАПИСЬ СТАТУСА (выполняется ВСЕГДА)
       // =================================================================
       #out_Status.PU_Total := #stat_PU_LastOut;

       IF #temp_PosActive > 0 THEN
           #out_Status.PU_Current_Avg := #temp_PU_Sum / INT_TO_REAL(#temp_PosActive);
       ELSE
           #out_Status.PU_Current_Avg := 0.0;
       END_IF;

       #out_Status.TempProd_Max := #temp_TempMax;
       #out_Status.Speed_Act := #inp_SpeedAct;
       #out_Status.PosCount := #temp_PosActive;
       #out_Status.Line_Run := #inp_LineRun;

       // =================================================================
       // 9. КОНТРОЛЬ ТЕМПЕРАТУРЫ ВОДЫ (ОТКЛОНЕНИЯ) - выполняется ВСЕГДА
       // =================================================================
       FOR #temp_PosIndex := 1 TO 9 DO
           #temp_TempDev := ABS(#ino_Recipe.ZoneConfig[#temp_PosIndex].TempWater_Set -
                                #inp_TempWater[#temp_PosIndex]);

           // Проверка отклонения от уставки
           IF #temp_TempDev > "DB_Config".c_MaxTempDev THEN
               #out_Alarm.Temp_Deviation := TRUE;
               #out_Alarm.Stop_Request := TRUE;
           END_IF;

           // Проверка датчика на обрыв/КЗ (выход за физически возможный диапазон)
           IF #inp_TempWater[#temp_PosIndex] < -10.0 OR #inp_TempWater[#temp_PosIndex] > 100.0 THEN
               #out_Alarm.Sensor_Fault := TRUE;
               #out_Alarm.Stop_Request := TRUE;
           END_IF;
       END_FOR;

       // =================================================================
       // 10. ФИНАЛЬНЫЙ СТАТУС
       // =================================================================
       #out_Alarm.Jam_Detected := #inp_Jam;
END_FUNCTION_BLOCK

FUNCTION_BLOCK "Расчет ПЕ по Зонам(aver)"   // FB32, SCL
{ S7_Optimized_Access := 'TRUE' }
VERSION : 0.1
   VAR_INPUT
      inp_Enable : Bool;   // Разрешение расчёта
      inp_bLineRun : Bool;   // Конвейер работает
      inp_bJam : Bool;   // Сигнал затора
      inp_SpeedAct : Real;   // Скорость ленты (м/мин)
      inp_TempWater : Array[1..9] of Real;   // Факт. T воды по зонам
      inp_ZonesConfig : Array[1..9] of "Zone_Config_V3";
   END_VAR
   VAR_OUTPUT
      out_Status : "Status_V3";   // Статус (DB174)
      out_Alarm : "Alarm";   // Аварии (DB175)
   END_VAR
   VAR_IN_OUT
      ino_StopMgr : "StopMgr";   // Менеджер остановок (DB176)
   END_VAR
   VAR
      stat_CycleTimer : IEC_TIMER;   // Таймер 1 секунда
      stat_PU_LastOut : Real;   // ПЕ последней вышедшей бутылки
      stat_TempProd_Current : Real;   // Текущая расчётная температура продукта (между зонами)
      stat_PU_Flow : Real;   // Средние ПЕ в потоке
      temp_PU_Total : Real;
      temp_TimeInZone : Real;   // Время в текущей зоне (мин)
      rStopDuration_Min : Real;   // Длительность простоя в минутах
      bCalcPositions : Bool;   // Флаг: выполнять ли расчёт движения
      temp_SourcePos : Int;   // Исходная позиция (сдвиг)
      temp_TempOut : Real;   // Т-ра продукта на выходе из зоны
      temp_TempAvg : Real;   // Средняя Т-ра в зоне
      temp_PU_Zone : Real;   // ПЕ для текущей зоны
   END_VAR
   VAR_TEMP
      temp_CycleTime_Min : Real;
      temp_PosIndex : Int;
      temp_ZoneIdx : Int;   // Время цикла (мин)
      temp_TempWater : Real;   // Счётчик позиций
      temp_DeltaT : Real;   // Исходная позиция (сдвиг)
      temp_PU_Inc : Real;   // Индекс зоны
      temp_TempMax : Real;   // T воды в текущей зоне
      temp_PU_Sum : Real;   // Изменение T продукта
      temp_PosActive : Int;   // Прирост ПЕ за цикл
      temp_TempDev : Real;   // Отклонение T воды
      temp_DistPerSec : Real;   // М/с дист за 1 сек
      temp_PosPerSec : Real;   // Кол-во активных позиций за 1 секунду
      temp_TempHotZones : Real;   // Отклонение T воды
   END_VAR
BEGIN

       // =================================================================
       // 1. ТАЙМЕР ЦИКЛА РАСЧЁТА (1 СЕКУНДА)
       // =================================================================

       #stat_CycleTimer.TON(IN := true, PT := t#1S);


       // Если 1 секунда ещё не прошла - выход из блока
       // 

       IF NOT #stat_CycleTimer.Q THEN
           RETURN;
       END_IF;

       // Сброс таймера для следующего цикла
       #stat_CycleTimer.TON(IN := FALSE, PT := t#0s);

       // Время цикла в минутах (для формулы ПЕ)
       #temp_CycleTime_Min := 1.0 / 60.0;

       // =================================================================
       // 2. ОБРАБОТКА ОСТАНОВКИ / ЗАТОРА
       // =================================================================
       // Флаг: можно ли выполнять расчёт движения
       #bCalcPositions := #inp_bLineRun AND NOT #inp_bJam;

       IF NOT #bCalcPositions THEN
           // === РЕЖИМ ПРОСТОЯ ===

           // Запуск таймера простоя
           #ino_StopMgr.Timer_Stop.TON(IN := TRUE,
                                       PT := T#100m,ET => #ino_StopMgr.Duration);

           // Преобразование времени: TIME -> DINT -> REAL -> минуты
           // TIME_TO_DINT возвращает миллисекунды как целое число
           #rStopDuration_Min := DINT_TO_REAL(TIME_TO_DINT(#ino_StopMgr.Duration)) / 60000.0;

           // Флаги для управления температурой и отбраковкой
           // 
           IF #rStopDuration_Min > "DB_Param_Calc_PE".cR_StopLimit_Short THEN  // > 2 минут
               #out_Alarm.Temp_Deviation := TRUE;  // ----Сигнал для снижения уставок!!! Привязать к блоку управления уставками Пастеризации
           END_IF;

           IF #rStopDuration_Min > "DB_Param_Calc_PE".cR_StopLimit_Long THEN  // > 5 минут
               #ino_StopMgr.Reject_Required := TRUE;
           END_IF;

           // Расчёт ПЕ во время простоя (горячие зоны 5-6)
           #temp_TempHotZones := (#inp_TempWater[5] + #inp_TempWater[6]) / 2.0;

           IF #temp_TempHotZones > "DB_Param_Calc_PE".cR_BaseTemp THEN
               //__________Расчет по формуле PUstop = ___________
               #ino_StopMgr.PU_Stop_Add :=
               #rStopDuration_Min *
               "DB_Param_Calc_PE".cR_Factor ** ((#temp_TempHotZones - "DB_Param_Calc_PE".cR_BaseTemp) / "DB_Param_Calc_PE".cR_Z_Value);
           ELSE
               #ino_StopMgr.PU_Stop_Add := 0.0;
           END_IF;

           // Пропускаем расчёт движения (код ниже выполнится только если #temp_CalcPositions = TRUE)
       ELSE
           // === РЕЖИМ РАБОТЫ ===

           // Линия работает - сброс таймера простоя
           #ino_StopMgr.Timer_Stop.TON(IN := FALSE, PT := t#0s);
           #ino_StopMgr.Duration := T#0s;
           #ino_StopMgr.PU_Stop_Add := 0.0;
           #out_Alarm.Temp_Deviation := FALSE;
       END_IF;

           // -------------------------------------------------------------
           // 3. РАСЧЁТ ПЕРЕМЕЩЕНИЯ ПРОДУКТА (ПОЗИЦИИ) 
           // -------------------------------------------------------------
           IF #bCalcPositions THEN

               // Проверка деления на ноль (защита от остановки при включенном флаге)
               IF #inp_SpeedAct <= 0.001 THEN
                   #out_Alarm.Stop_Request := TRUE;
                   RETURN;
               END_IF;

               // Инициализация: температура продукта на ВХОДЕ в туннель (из рецепта/оператора)
               #stat_TempProd_Current := "DB_Param_Calc_PE".cR_TempProd_Inlet;

               // Сброс накопленных ПЕ для текущего расчёта
               #temp_PU_Total := 0.0;

               // Цикл по всем 9 зонам
               FOR #temp_ZoneIdx := 1 TO 9 DO

                   // --- А. Расчёт времени пребывания в зоне ---
                   #temp_TimeInZone := #inp_ZonesConfig[#temp_ZoneIdx].Length / #inp_SpeedAct;

                   // Сохраняем время в структуру статуса для HMI
                   #out_Status.ZoneData[#temp_ZoneIdx].TimeInZone := #temp_TimeInZone;
                   #out_Status.ZoneData[#temp_ZoneIdx].TempWater_Act := #inp_TempWater[#temp_ZoneIdx];

                   // --- Б. Расчёт температуры продукта НА ВЫХОДЕ из зоны ---
                   // Формула: T_out = T_water - (T_water - T_in) * e^(-K * t)
                   // Используем EXP() для числа Эйлера
                   #temp_TempOut := #inp_TempWater[#temp_ZoneIdx] -
                   (#inp_TempWater[#temp_ZoneIdx] - #stat_TempProd_Current) *
                   EXP(- "DB_Param_Calc_PE".cR_K_Coeff * #temp_TimeInZone);


                   // Сохраняем температуры в статус
                   #out_Status.ZoneData[#temp_ZoneIdx].TempProd_In := #stat_TempProd_Current;
                   #out_Status.ZoneData[#temp_ZoneIdx].TempProd_Out := #temp_TempOut;

                   // --- В. Расчёт средней температуры в зоне ---
                   #temp_TempAvg := (#stat_TempProd_Current + #temp_TempOut) / 2.0;
                   #out_Status.ZoneData[#temp_ZoneIdx].TempProd_Avg := #temp_TempAvg;

                   // --- Г. Расчёт ПЕ для зоны ---
                   // ПЕ копятся только если средняя температура >= 60°C
                   IF #temp_TempAvg >= "DB_Param_Calc_PE".cR_BaseTemp THEN
                       #temp_PU_Zone := #temp_TimeInZone *
                       "DB_Param_Calc_PE".cR_Factor **
                       ((#temp_TempAvg - "DB_Param_Calc_PE".cR_BaseTemp) / "DB_Param_Calc_PE".cR_Z_Value);
                   ELSE
                       #temp_PU_Zone := 0.0;
                   END_IF;

                   #out_Status.ZoneData[#temp_ZoneIdx].PU_Zone := #temp_PU_Zone;

                   // --- Д. Накопление итогов ---
                   #temp_PU_Total := #temp_PU_Total + #temp_PU_Zone;

                   // Подготовка температуры для следующей зоны: выход из текущей = вход в следующую
                   #stat_TempProd_Current := #temp_TempOut;

               END_FOR; // Конец цикла по зонам

               // Сохраняем температуру выхода из туннеля
               #out_Status.TempProd_Exit := #stat_TempProd_Current;

               // =================================================================
               // 4. ФИНАЛИЗАЦИЯ РАСЧЁТА
               // =================================================================

               // Итоговые ПЕ = ПЕ потока + ПЕ простоя (если были)
               #out_Status.PU_Total := #temp_PU_Total + #ino_StopMgr.PU_Stop_Add;

               // Сохраняем значение для истории (последняя вышедшая партия)
               #stat_PU_LastOut := #out_Status.PU_Total;

               // Проверка качества (Уставки из рецепта)
               IF #out_Status.PU_Total < "DB_Param_Calc_PE".cR_PU_Target_Min THEN
                   #out_Alarm.PU_Under := TRUE;
                   #out_Alarm.Stop_Request := TRUE;
               ELSE
                   #out_Alarm.PU_Under := FALSE;
               END_IF;

               IF #out_Status.PU_Total > "DB_Param_Calc_PE".cR_PU_Target_Max THEN
                   #out_Alarm.PU_Over := TRUE;
                   #out_Alarm.Stop_Request := TRUE;
               ELSE
                   #out_Alarm.PU_Over := FALSE;
               END_IF;

               #out_Status.Calculation_Ready := TRUE;

           ELSE
               // Если линия стоит, сбрасываем флаг готовности, но сохраняем последние значения
               #out_Status.Calculation_Ready := FALSE;
           END_IF;

           // =================================================================
           // 5. КОНТРОЛЬ ДАТЧИКОВ И АВАРИИ (Вне зависимости от режима)
           // =================================================================
           #out_Status.Speed_Act := #inp_SpeedAct;
           #out_Status.Line_Run := #inp_bLineRun;
           #out_Alarm.Jam_Detected := #inp_bJam;

           FOR #temp_ZoneIdx := 1 TO 9 DO
               // Проверка отклонения от уставки
               #temp_TempDev := ABS(#inp_ZonesConfig[#temp_ZoneIdx].TempWater_Set -
                                    #inp_TempWater[#temp_ZoneIdx]);

               IF #temp_TempDev > "DB_Param_Calc_PE".cR_MaxTempDev THEN
                   #out_Alarm.Temp_Deviation := TRUE;
                   #out_Alarm.Stop_Request := TRUE;
               END_IF;
           END_FOR;
END_FUNCTION_BLOCK

FUNCTION_BLOCK "FB_Convert_For_RS485"   // FB33, SCL
{ S7_Optimized_Access := 'TRUE' }
VERSION : 0.1
   VAR_INPUT
      iSet_Pos : Int;   // Входное значение для регул клапана
   END_VAR
   VAR_OUTPUT
      iOutPosForRS_485 : Int;
   END_VAR
   VAR_TEMP
      rConvertNum : Real;   // Значение конвертированное в Реал
   END_VAR
BEGIN

   //_____Ковертация входного значения в реал для расчета без потери десяток___
   //
   #rConvertNum := INT_TO_REAL(#iSet_Pos);

   // Обратное преобразование в инт с делением на
   // 2.7648 - это значение выхода для АЦП - преобразуем его в 0-100%

   #iOutPosForRS_485 := REAL_TO_INT(IN := #rConvertNum / 2.7648);
END_FUNCTION_BLOCK

FUNCTION "Клапана_О/З" : Void   // FC1, LAD
{ S7_Optimized_Access := 'TRUE' }
VERSION : 0.1
BEGIN

REGION Network 1: Клапан Химия - 1
   // Клапан Химия - 1
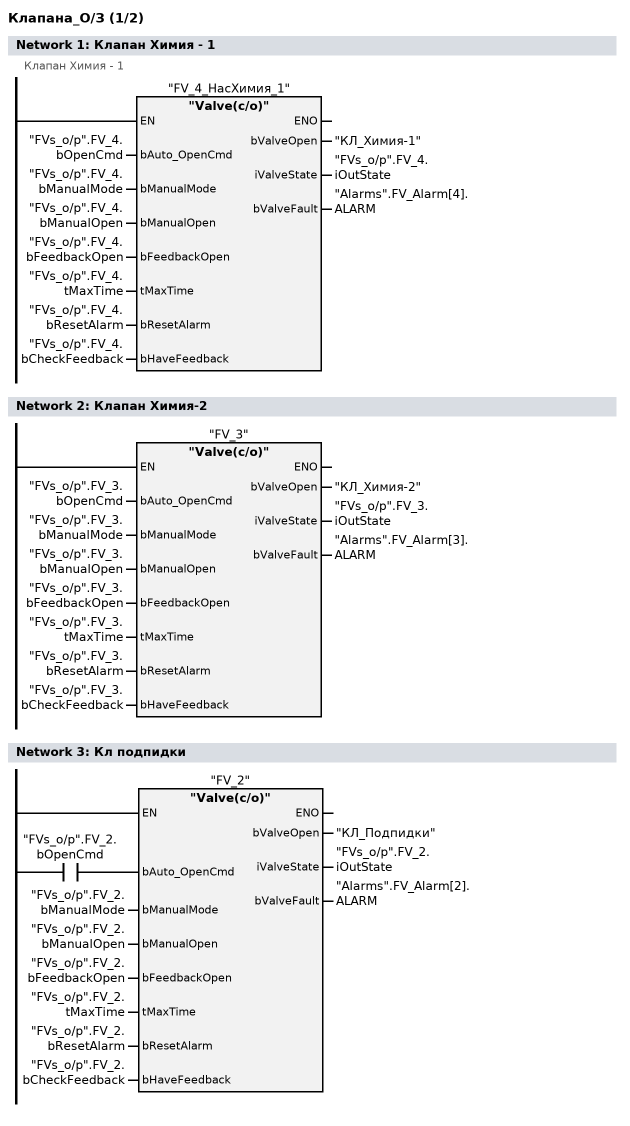
   RUNG wire#powerrail
      "FV_4_НасХимия_1"(bAuto_OpenCmd := "FVs_o/p".FV_4.bOpenCmd, bManualMode := "FVs_o/p".FV_4.bManualMode, bManualOpen := "FVs_o/p".FV_4.bManualOpen, bFeedbackOpen := "FVs_o/p".FV_4.bFeedbackOpen, tMaxTime := "FVs_o/p".FV_4.tMaxTime, bResetAlarm := "FVs_o/p".FV_4.bResetAlarm, bHaveFeedback := "FVs_o/p".FV_4.bCheckFeedback, bValveOpen => "КЛ_Химия-1", iValveState => "FVs_o/p".FV_4.iOutState, bValveFault => "Alarms".FV_Alarm[4].ALARM)
   END_RUNG
   // the same network as SCL:
   "FV_4_НасХимия_1"(bAuto_OpenCmd := "FVs_o/p".FV_4.bOpenCmd,   // "Valve(c/o)"
                     bManualMode := "FVs_o/p".FV_4.bManualMode,
                     bManualOpen := "FVs_o/p".FV_4.bManualOpen,
                     bFeedbackOpen := "FVs_o/p".FV_4.bFeedbackOpen,
                     tMaxTime := "FVs_o/p".FV_4.tMaxTime,
                     bResetAlarm := "FVs_o/p".FV_4.bResetAlarm,
                     bHaveFeedback := "FVs_o/p".FV_4.bCheckFeedback,
                     bValveOpen => "КЛ_Химия-1",
                     iValveState => "FVs_o/p".FV_4.iOutState,
                     bValveFault => "Alarms".FV_Alarm[4].ALARM);
END_REGION

REGION Network 2: Клапан Химия-2
   RUNG wire#powerrail
      "FV_3"(bAuto_OpenCmd := "FVs_o/p".FV_3.bOpenCmd, bManualMode := "FVs_o/p".FV_3.bManualMode, bManualOpen := "FVs_o/p".FV_3.bManualOpen, bFeedbackOpen := "FVs_o/p".FV_3.bFeedbackOpen, tMaxTime := "FVs_o/p".FV_3.tMaxTime, bResetAlarm := "FVs_o/p".FV_3.bResetAlarm, bHaveFeedback := "FVs_o/p".FV_3.bCheckFeedback, bValveOpen => "КЛ_Химия-2", iValveState => "FVs_o/p".FV_3.iOutState, bValveFault => "Alarms".FV_Alarm[3].ALARM)
   END_RUNG
   // the same network as SCL:
   "FV_3"(bAuto_OpenCmd := "FVs_o/p".FV_3.bOpenCmd,   // "Valve(c/o)"
          bManualMode := "FVs_o/p".FV_3.bManualMode,
          bManualOpen := "FVs_o/p".FV_3.bManualOpen,
          bFeedbackOpen := "FVs_o/p".FV_3.bFeedbackOpen,
          tMaxTime := "FVs_o/p".FV_3.tMaxTime,
          bResetAlarm := "FVs_o/p".FV_3.bResetAlarm,
          bHaveFeedback := "FVs_o/p".FV_3.bCheckFeedback,
          bValveOpen => "КЛ_Химия-2",
          iValveState => "FVs_o/p".FV_3.iOutState,
          bValveFault => "Alarms".FV_Alarm[3].ALARM);
END_REGION

REGION Network 3: Кл подпидки
   RUNG wire#powerrail
      "FV_2"(bAuto_OpenCmd := wire#w1, bManualMode := "FVs_o/p".FV_2.bManualMode, bManualOpen := "FVs_o/p".FV_2.bManualOpen, bFeedbackOpen := "FVs_o/p".FV_2.bFeedbackOpen, tMaxTime := "FVs_o/p".FV_2.tMaxTime, bResetAlarm := "FVs_o/p".FV_2.bResetAlarm, bHaveFeedback := "FVs_o/p".FV_2.bCheckFeedback, bValveOpen => "КЛ_Подпидки", iValveState => "FVs_o/p".FV_2.iOutState, bValveFault => "Alarms".FV_Alarm[2].ALARM)
   END_RUNG
   RUNG wire#powerrail
      Contact( "FVs_o/p".FV_2.bOpenCmd )
   END_RUNG wire#w1
   // the same network as SCL:
   "FV_2"(bAuto_OpenCmd := "FVs_o/p".FV_2.bOpenCmd,   // "Valve(c/o)"
          bManualMode := "FVs_o/p".FV_2.bManualMode,
          bManualOpen := "FVs_o/p".FV_2.bManualOpen,
          bFeedbackOpen := "FVs_o/p".FV_2.bFeedbackOpen,
          tMaxTime := "FVs_o/p".FV_2.tMaxTime,
          bResetAlarm := "FVs_o/p".FV_2.bResetAlarm,
          bHaveFeedback := "FVs_o/p".FV_2.bCheckFeedback,
          bValveOpen => "КЛ_Подпидки",
          iValveState => "FVs_o/p".FV_2.iOutState,
          bValveFault => "Alarms".FV_Alarm[2].ALARM);
END_REGION

REGION Network 4: Клапан пара
   // Пара
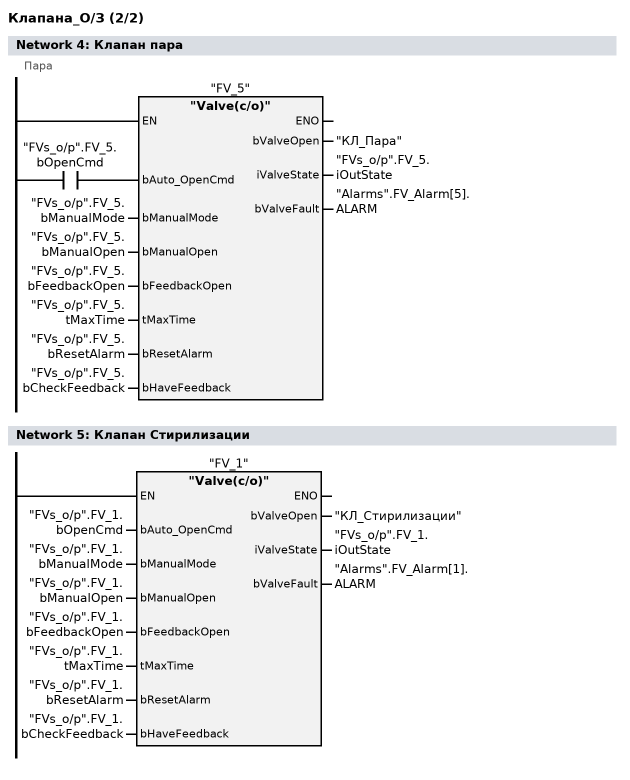
   RUNG wire#powerrail
      "FV_5"(bAuto_OpenCmd := wire#w1, bManualMode := "FVs_o/p".FV_5.bManualMode, bManualOpen := "FVs_o/p".FV_5.bManualOpen, bFeedbackOpen := "FVs_o/p".FV_5.bFeedbackOpen, tMaxTime := "FVs_o/p".FV_5.tMaxTime, bResetAlarm := "FVs_o/p".FV_5.bResetAlarm, bHaveFeedback := "FVs_o/p".FV_5.bCheckFeedback, bValveOpen => "КЛ_Пара", iValveState => "FVs_o/p".FV_5.iOutState, bValveFault => "Alarms".FV_Alarm[5].ALARM)
   END_RUNG
   RUNG wire#powerrail
      Contact( "FVs_o/p".FV_5.bOpenCmd )
   END_RUNG wire#w1
   // the same network as SCL:
   "FV_5"(bAuto_OpenCmd := "FVs_o/p".FV_5.bOpenCmd,   // "Valve(c/o)"
          bManualMode := "FVs_o/p".FV_5.bManualMode,
          bManualOpen := "FVs_o/p".FV_5.bManualOpen,
          bFeedbackOpen := "FVs_o/p".FV_5.bFeedbackOpen,
          tMaxTime := "FVs_o/p".FV_5.tMaxTime,
          bResetAlarm := "FVs_o/p".FV_5.bResetAlarm,
          bHaveFeedback := "FVs_o/p".FV_5.bCheckFeedback,
          bValveOpen => "КЛ_Пара",
          iValveState => "FVs_o/p".FV_5.iOutState,
          bValveFault => "Alarms".FV_Alarm[5].ALARM);
END_REGION

REGION Network 5: Клапан Стирилизации
   RUNG wire#powerrail
      "FV_1"(bAuto_OpenCmd := "FVs_o/p".FV_1.bOpenCmd, bManualMode := "FVs_o/p".FV_1.bManualMode, bManualOpen := "FVs_o/p".FV_1.bManualOpen, bFeedbackOpen := "FVs_o/p".FV_1.bFeedbackOpen, tMaxTime := "FVs_o/p".FV_1.tMaxTime, bResetAlarm := "FVs_o/p".FV_1.bResetAlarm, bHaveFeedback := "FVs_o/p".FV_1.bCheckFeedback, bValveOpen => "КЛ_Стирилизации", iValveState => "FVs_o/p".FV_1.iOutState, bValveFault => "Alarms".FV_Alarm[1].ALARM)
   END_RUNG
   // the same network as SCL:
   "FV_1"(bAuto_OpenCmd := "FVs_o/p".FV_1.bOpenCmd,   // "Valve(c/o)"
          bManualMode := "FVs_o/p".FV_1.bManualMode,
          bManualOpen := "FVs_o/p".FV_1.bManualOpen,
          bFeedbackOpen := "FVs_o/p".FV_1.bFeedbackOpen,
          tMaxTime := "FVs_o/p".FV_1.tMaxTime,
          bResetAlarm := "FVs_o/p".FV_1.bResetAlarm,
          bHaveFeedback := "FVs_o/p".FV_1.bCheckFeedback,
          bValveOpen => "КЛ_Стирилизации",
          iValveState => "FVs_o/p".FV_1.iOutState,
          bValveFault => "Alarms".FV_Alarm[1].ALARM);
END_REGION
END_FUNCTION

FUNCTION "Клапана_Регул" : Void   // FC2, LAD
{ S7_Optimized_Access := 'TRUE' }
VERSION : 0.1
BEGIN

